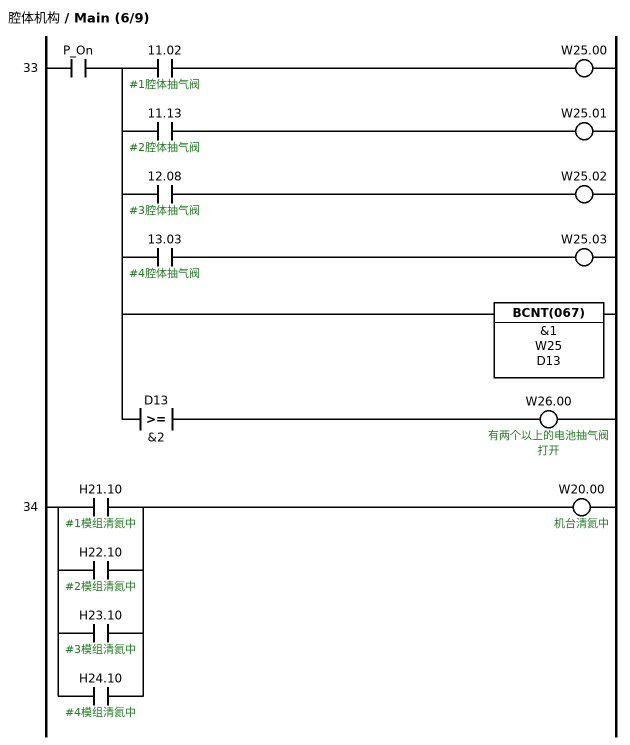
; [picture p240: 腔体机构 / Main, rungs 33-34]
; rung 33
LD P_On
OUT TR0
AND 11.02  ; #1腔体抽气阀
OUT W25.00
LD TR0
AND 11.13  ; #2腔体抽气阀
OUT W25.01
LD TR0
AND 12.08  ; #3腔体抽气阀
OUT W25.02
LD TR0
AND 13.03  ; #4腔体抽气阀
OUT W25.03
LD TR0
BCNT(067) &1 W25 D13
AND>=(325) D13 &2
OUT W26.00  ; 有两个以上的电池抽气阀打开
; rung 34
LD H21.10  ; #1模组清氦中
OR H22.10  ; #2模组清氦中
OR H23.10  ; #3模组清氦中
OR H24.10  ; #4模组清氦中
OUT W20.00  ; 机台清氦中

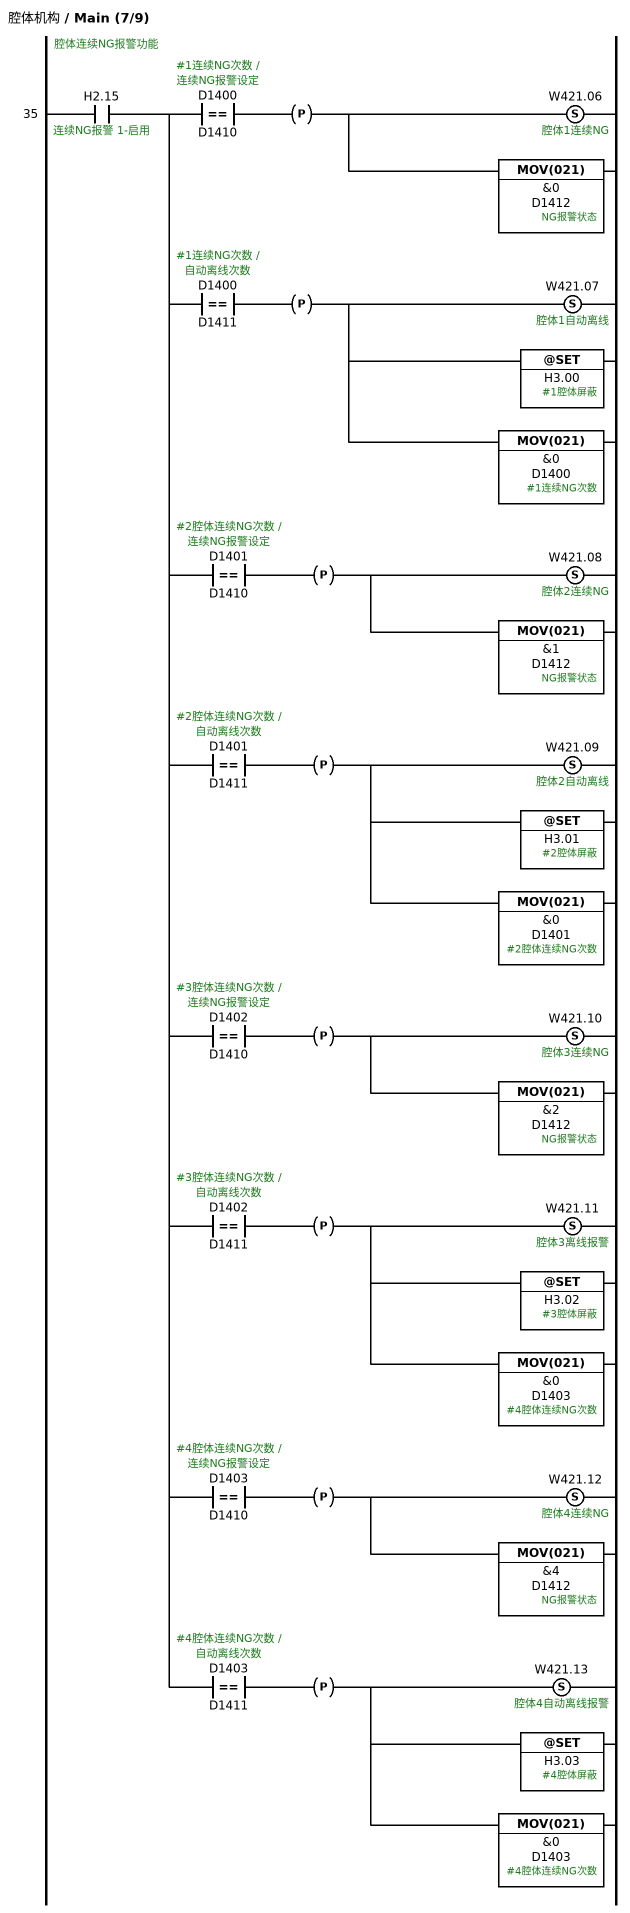
; rung 35: 腔体连续NG报警功能
LD H2.15  ; 连续NG报警 1-启用
OUT TR0
AND=(300) D1400 D1410  ; #1连续NG次数, 连续NG报警设定
UP(521)
SET W421.06  ; 腔体1连续NG
MOV(021) &0 D1412  ; NG报警状态
LD TR0
AND=(300) D1400 D1411  ; #1连续NG次数, 自动离线次数
UP(521)
SET W421.07  ; 腔体1自动离线
@SET H3.00  ; #1腔体屏蔽
MOV(021) &0 D1400  ; #1连续NG次数
LD TR0
AND=(300) D1401 D1410  ; #2腔体连续NG次数, 连续NG报警设定
UP(521)
SET W421.08  ; 腔体2连续NG
MOV(021) &1 D1412  ; NG报警状态
LD TR0
AND=(300) D1401 D1411  ; #2腔体连续NG次数, 自动离线次数
UP(521)
SET W421.09  ; 腔体2自动离线
@SET H3.01  ; #2腔体屏蔽
MOV(021) &0 D1401  ; #2腔体连续NG次数
LD TR0
AND=(300) D1402 D1410  ; #3腔体连续NG次数, 连续NG报警设定
UP(521)
SET W421.10  ; 腔体3连续NG
MOV(021) &2 D1412  ; NG报警状态
LD TR0
AND=(300) D1402 D1411  ; #3腔体连续NG次数, 自动离线次数
UP(521)
SET W421.11  ; 腔体3离线报警
@SET H3.02  ; #3腔体屏蔽
MOV(021) &0 D1403  ; #4腔体连续NG次数
LD TR0
AND=(300) D1403 D1410  ; #4腔体连续NG次数, 连续NG报警设定
UP(521)
SET W421.12  ; 腔体4连续NG
MOV(021) &4 D1412  ; NG报警状态
LD TR0
AND=(300) D1403 D1411  ; #4腔体连续NG次数, 自动离线次数
UP(521)
SET W421.13  ; 腔体4自动离线报警
@SET H3.03  ; #4腔体屏蔽
MOV(021) &0 D1403  ; #4腔体连续NG次数

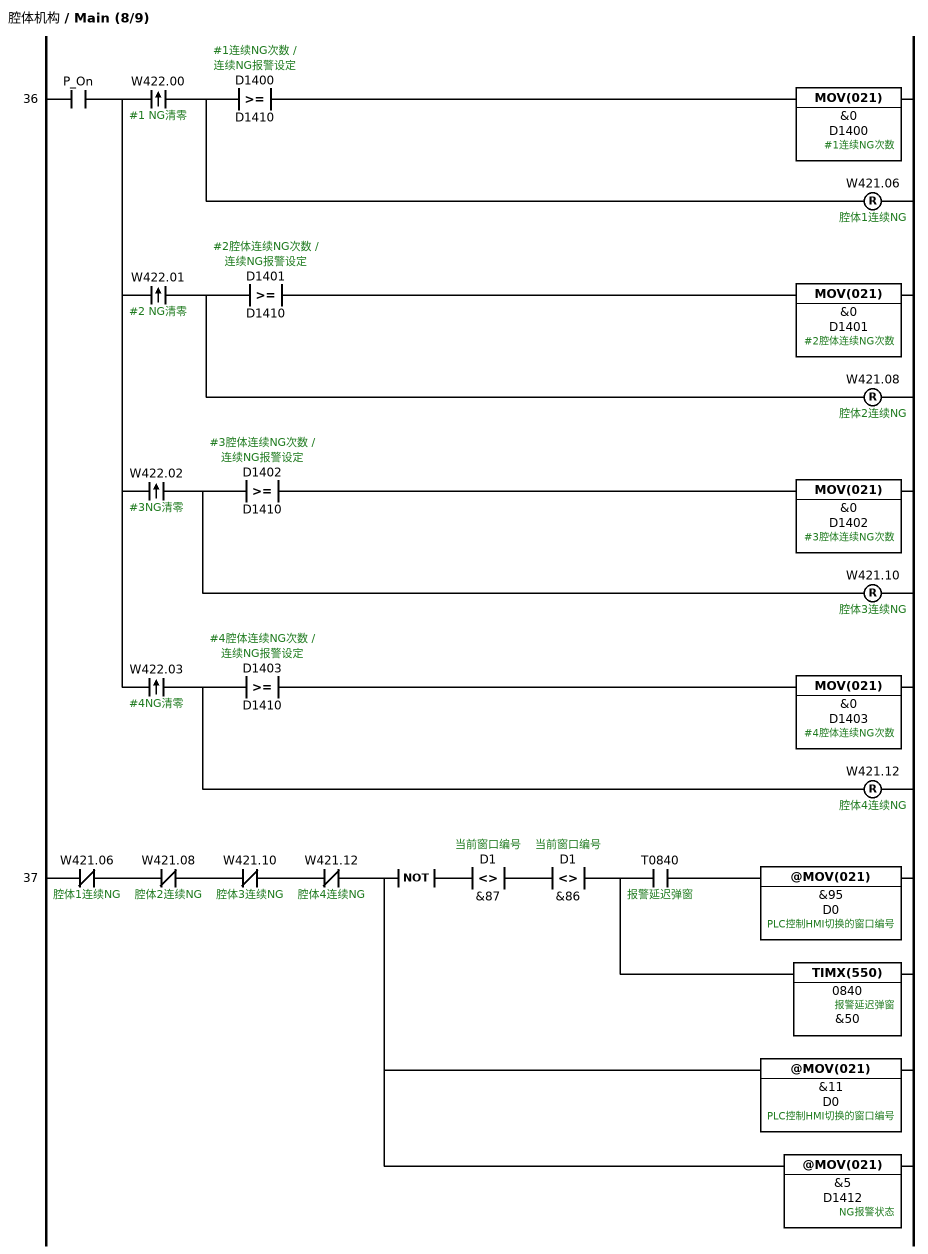
; rung 36
LD P_On
OUT TR0
@AND W422.00  ; #1 NG清零
OUT TR1
AND>=(325) D1400 D1410  ; #1连续NG次数, 连续NG报警设定
MOV(021) &0 D1400  ; #1连续NG次数
LD TR1
RSET W421.06  ; 腔体1连续NG
LD TR0
@AND W422.01  ; #2 NG清零
OUT TR1
AND>=(325) D1401 D1410  ; #2腔体连续NG次数, 连续NG报警设定
MOV(021) &0 D1401  ; #2腔体连续NG次数
LD TR1
RSET W421.08  ; 腔体2连续NG
LD TR0
@AND W422.02  ; #3NG清零
OUT TR1
AND>=(325) D1402 D1410  ; #3腔体连续NG次数, 连续NG报警设定
MOV(021) &0 D1402  ; #3腔体连续NG次数
LD TR1
RSET W421.10  ; 腔体3连续NG
LD TR0
@AND W422.03  ; #4NG清零
OUT TR0
AND>=(325) D1403 D1410  ; #4腔体连续NG次数, 连续NG报警设定
MOV(021) &0 D1403  ; #4腔体连续NG次数
LD TR0
RSET W421.12  ; 腔体4连续NG
; rung 37
LDNOT W421.06  ; 腔体1连续NG
ANDNOT W421.08  ; 腔体2连续NG
ANDNOT W421.10  ; 腔体3连续NG
ANDNOT W421.12  ; 腔体4连续NG
OUT TR0
NOT(520)
AND<>(305) D1 &87  ; 当前窗口编号
AND<>(305) D1 &86  ; 当前窗口编号
OUT TR1
AND T0840  ; 报警延迟弹窗
@MOV(021) &95 D0  ; PLC控制HMI切换的窗口编号
LD TR1
TIMX(550) 0840 &50  ; 报警延迟弹窗
LD TR0
@MOV(021) &11 D0  ; PLC控制HMI切换的窗口编号
@MOV(021) &5 D1412  ; NG报警状态

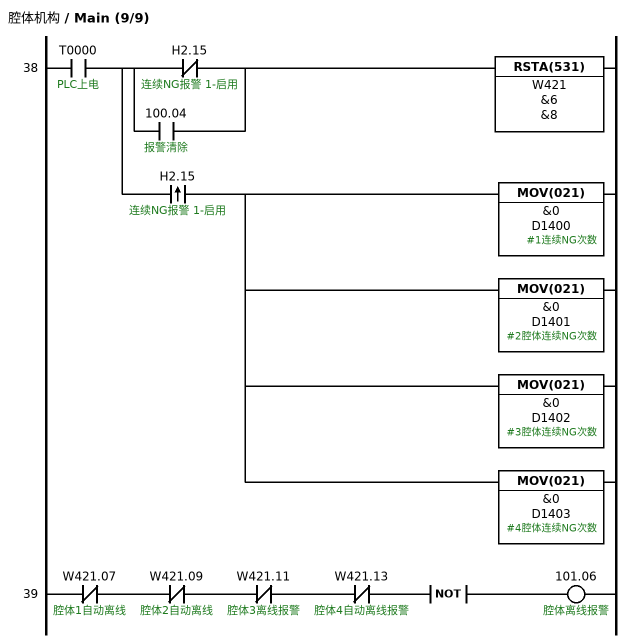
; rung 38
LD T0000  ; PLC上电
OUT TR0
LDNOT H2.15  ; 连续NG报警 1-启用
OR 100.04  ; 报警清除
ANDLD
RSTA(531) W421 &6 &8
LD TR0
@AND H2.15  ; 连续NG报警 1-启用
MOV(021) &0 D1400  ; #1连续NG次数
MOV(021) &0 D1401  ; #2腔体连续NG次数
MOV(021) &0 D1402  ; #3腔体连续NG次数
MOV(021) &0 D1403  ; #4腔体连续NG次数
; rung 39
LDNOT W421.07  ; 腔体1自动离线
ANDNOT W421.09  ; 腔体2自动离线
ANDNOT W421.11  ; 腔体3离线报警
ANDNOT W421.13  ; 腔体4自动离线报警
NOT(520)
OUT 101.06  ; 腔体离线报警

### Section 工站复位

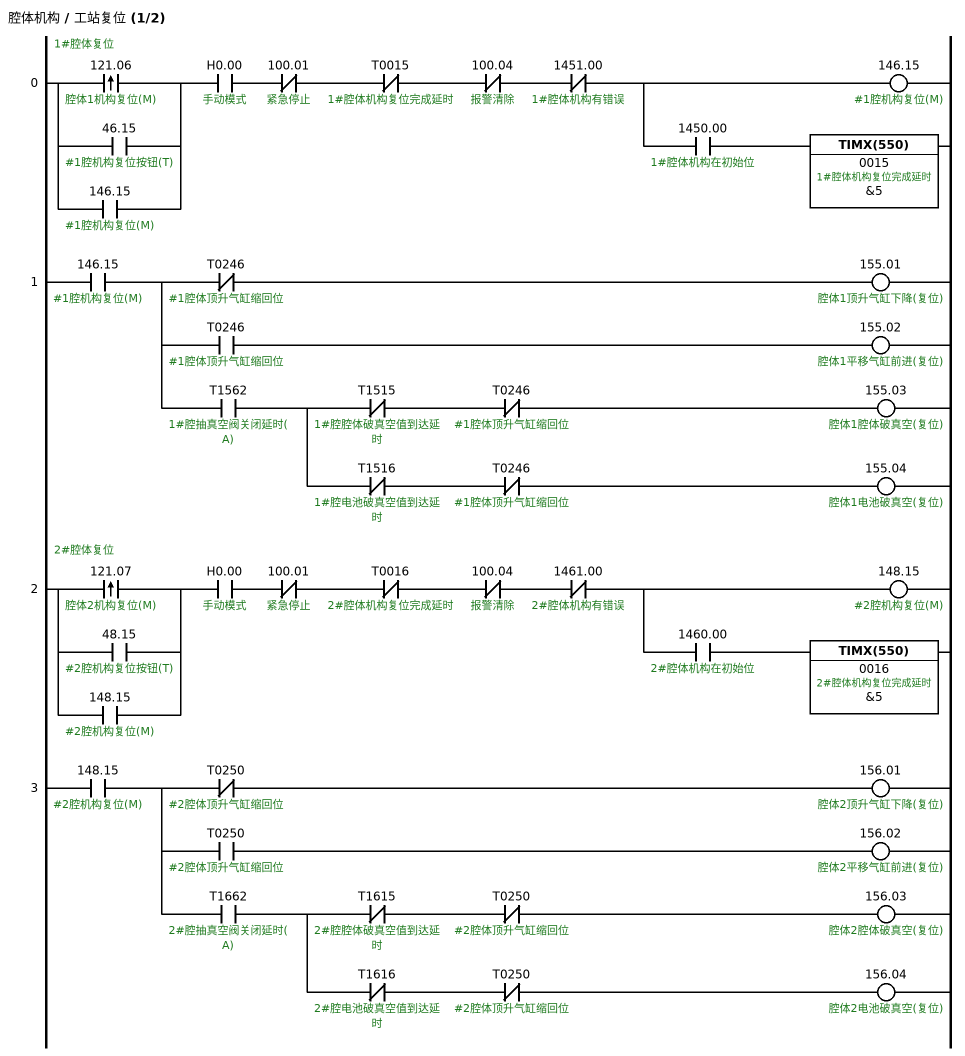
; rung 0: 1#腔体复位
@LD 121.06  ; 腔体1机构复位(M)
OR 46.15  ; #1腔机构复位按钮(T)
OR 146.15  ; #1腔机构复位(M)
AND H0.00  ; 手动模式
ANDNOT 100.01  ; 紧急停止
ANDNOT T0015  ; 1#腔体机构复位完成延时
ANDNOT 100.04  ; 报警清除
ANDNOT 1451.00  ; 1#腔体机构有错误
OUT 146.15  ; #1腔机构复位(M)
AND 1450.00  ; 1#腔体机构在初始位
TIMX(550) 0015 &5  ; 1#腔体机构复位完成延时
; rung 1
LD 146.15  ; #1腔机构复位(M)
OUT TR0
ANDNOT T0246  ; #1腔体顶升气缸缩回位
OUT 155.01  ; 腔体1顶升气缸下降(复位)
LD TR0
AND T0246  ; #1腔体顶升气缸缩回位
OUT 155.02  ; 腔体1平移气缸前进(复位)
LD TR0
AND T1562  ; 1#腔抽真空阀关闭延时(A)
OUT TR0
ANDNOT T1515  ; 1#腔腔体破真空值到达延时
ANDNOT T0246  ; #1腔体顶升气缸缩回位
OUT 155.03  ; 腔体1腔体破真空(复位)
LD TR0
ANDNOT T1516  ; 1#腔电池破真空值到达延时
ANDNOT T0246  ; #1腔体顶升气缸缩回位
OUT 155.04  ; 腔体1电池破真空(复位)
; rung 2: 2#腔体复位
@LD 121.07  ; 腔体2机构复位(M)
OR 48.15  ; #2腔机构复位按钮(T)
OR 148.15  ; #2腔机构复位(M)
AND H0.00  ; 手动模式
ANDNOT 100.01  ; 紧急停止
ANDNOT T0016  ; 2#腔体机构复位完成延时
ANDNOT 100.04  ; 报警清除
ANDNOT 1461.00  ; 2#腔体机构有错误
OUT 148.15  ; #2腔机构复位(M)
AND 1460.00  ; 2#腔体机构在初始位
TIMX(550) 0016 &5  ; 2#腔体机构复位完成延时
; rung 3
LD 148.15  ; #2腔机构复位(M)
OUT TR0
ANDNOT T0250  ; #2腔体顶升气缸缩回位
OUT 156.01  ; 腔体2顶升气缸下降(复位)
LD TR0
AND T0250  ; #2腔体顶升气缸缩回位
OUT 156.02  ; 腔体2平移气缸前进(复位)
LD TR0
AND T1662  ; 2#腔抽真空阀关闭延时(A)
OUT TR0
ANDNOT T1615  ; 2#腔腔体破真空值到达延时
ANDNOT T0250  ; #2腔体顶升气缸缩回位
OUT 156.03  ; 腔体2腔体破真空(复位)
LD TR0
ANDNOT T1616  ; 2#腔电池破真空值到达延时
ANDNOT T0250  ; #2腔体顶升气缸缩回位
OUT 156.04  ; 腔体2电池破真空(复位)

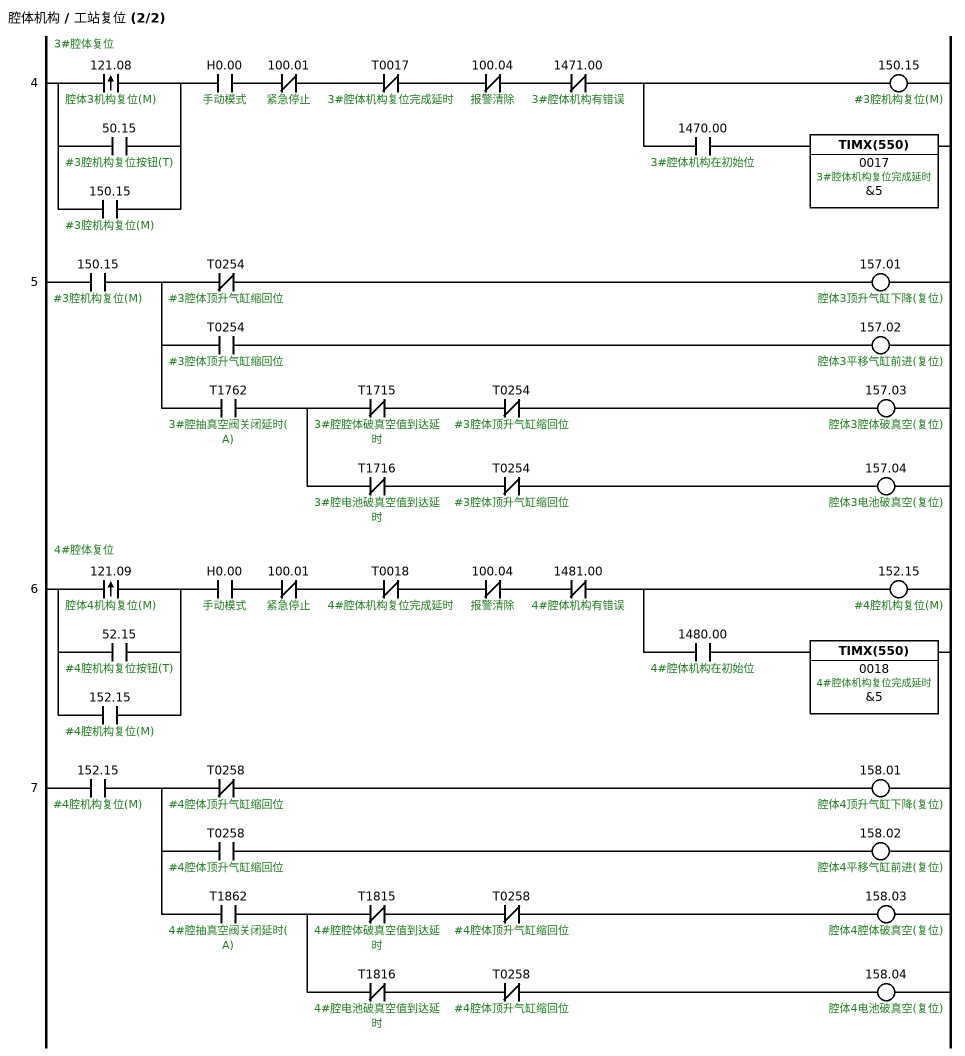
; rung 4: 3#腔体复位
@LD 121.08  ; 腔体3机构复位(M)
OR 50.15  ; #3腔机构复位按钮(T)
OR 150.15  ; #3腔机构复位(M)
AND H0.00  ; 手动模式
ANDNOT 100.01  ; 紧急停止
ANDNOT T0017  ; 3#腔体机构复位完成延时
ANDNOT 100.04  ; 报警清除
ANDNOT 1471.00  ; 3#腔体机构有错误
OUT 150.15  ; #3腔机构复位(M)
AND 1470.00  ; 3#腔体机构在初始位
TIMX(550) 0017 &5  ; 3#腔体机构复位完成延时
; rung 5
LD 150.15  ; #3腔机构复位(M)
OUT TR0
ANDNOT T0254  ; #3腔体顶升气缸缩回位
OUT 157.01  ; 腔体3顶升气缸下降(复位)
LD TR0
AND T0254  ; #3腔体顶升气缸缩回位
OUT 157.02  ; 腔体3平移气缸前进(复位)
LD TR0
AND T1762  ; 3#腔抽真空阀关闭延时(A)
OUT TR0
ANDNOT T1715  ; 3#腔腔体破真空值到达延时
ANDNOT T0254  ; #3腔体顶升气缸缩回位
OUT 157.03  ; 腔体3腔体破真空(复位)
LD TR0
ANDNOT T1716  ; 3#腔电池破真空值到达延时
ANDNOT T0254  ; #3腔体顶升气缸缩回位
OUT 157.04  ; 腔体3电池破真空(复位)
; rung 6: 4#腔体复位
@LD 121.09  ; 腔体4机构复位(M)
OR 52.15  ; #4腔机构复位按钮(T)
OR 152.15  ; #4腔机构复位(M)
AND H0.00  ; 手动模式
ANDNOT 100.01  ; 紧急停止
ANDNOT T0018  ; 4#腔体机构复位完成延时
ANDNOT 100.04  ; 报警清除
ANDNOT 1481.00  ; 4#腔体机构有错误
OUT 152.15  ; #4腔机构复位(M)
AND 1480.00  ; 4#腔体机构在初始位
TIMX(550) 0018 &5  ; 4#腔体机构复位完成延时
; rung 7
LD 152.15  ; #4腔机构复位(M)
OUT TR0
ANDNOT T0258  ; #4腔体顶升气缸缩回位
OUT 158.01  ; 腔体4顶升气缸下降(复位)
LD TR0
AND T0258  ; #4腔体顶升气缸缩回位
OUT 158.02  ; 腔体4平移气缸前进(复位)
LD TR0
AND T1862  ; 4#腔抽真空阀关闭延时(A)
OUT TR0
ANDNOT T1815  ; 4#腔腔体破真空值到达延时
ANDNOT T0258  ; #4腔体顶升气缸缩回位
OUT 158.03  ; 腔体4腔体破真空(复位)
LD TR0
ANDNOT T1816  ; 4#腔电池破真空值到达延时
ANDNOT T0258  ; #4腔体顶升气缸缩回位
OUT 158.04  ; 腔体4电池破真空(复位)

### Section _1_腔体手动

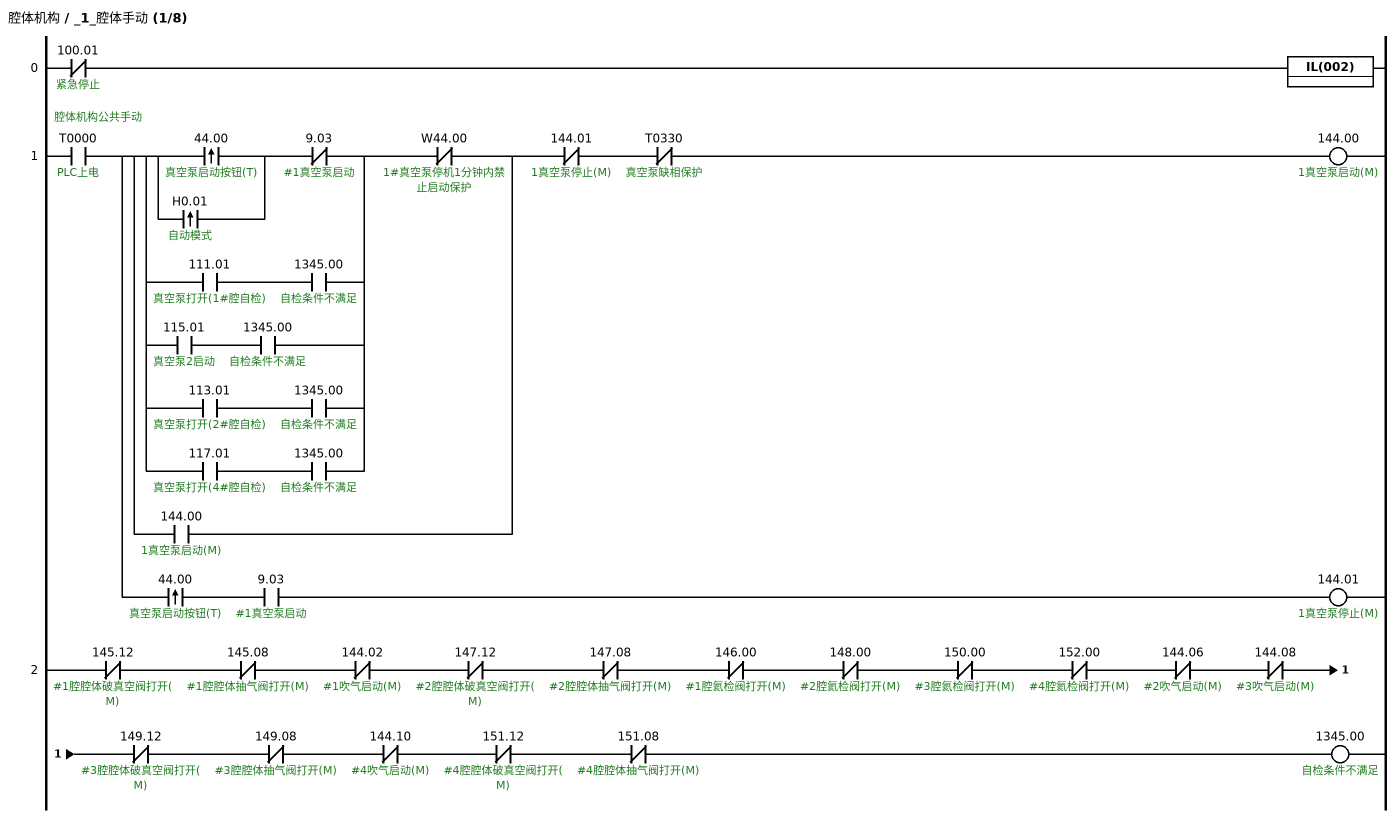
; rung 0
LDNOT 100.01  ; 紧急停止
IL(002)
; rung 1: 腔体机构公共手动
LD T0000  ; PLC上电
OUT TR0
@LD 44.00  ; 真空泵启动按钮(T)
@OR H0.01  ; 自动模式
ANDNOT 9.03  ; #1真空泵启动
LD 111.01  ; 真空泵打开(1#腔自检)
AND 1345.00  ; 自检条件不满足
ORLD
LD 115.01  ; 真空泵2启动
AND 1345.00  ; 自检条件不满足
ORLD
LD 113.01  ; 真空泵打开(2#腔自检)
AND 1345.00  ; 自检条件不满足
ORLD
LD 117.01  ; 真空泵打开(4#腔自检)
AND 1345.00  ; 自检条件不满足
ORLD
ANDNOT W44.00  ; 1#真空泵停机1分钟内禁止启动保护
OR 144.00  ; 1真空泵启动(M)
ANDLD
ANDNOT 144.01  ; 1真空泵停止(M)
ANDNOT T0330  ; 真空泵缺相保护
OUT 144.00  ; 1真空泵启动(M)
LD TR0
@AND 44.00  ; 真空泵启动按钮(T)
AND 9.03  ; #1真空泵启动
OUT 144.01  ; 1真空泵停止(M)
; rung 2
LDNOT 145.12  ; #1腔腔体破真空阀打开(M)
ANDNOT 145.08  ; #1腔腔体抽气阀打开(M)
ANDNOT 144.02  ; #1吹气启动(M)
ANDNOT 147.12  ; #2腔腔体破真空阀打开(M)
ANDNOT 147.08  ; #2腔腔体抽气阀打开(M)
ANDNOT 146.00  ; #1腔氦检阀打开(M)
ANDNOT 148.00  ; #2腔氦检阀打开(M)
ANDNOT 150.00  ; #3腔氦检阀打开(M)
ANDNOT 152.00  ; #4腔氦检阀打开(M)
ANDNOT 144.06  ; #2吹气启动(M)
ANDNOT 144.08  ; #3吹气启动(M)
ANDNOT 149.12  ; #3腔腔体破真空阀打开(M)
ANDNOT 149.08  ; #3腔腔体抽气阀打开(M)
ANDNOT 144.10  ; #4吹气启动(M)
ANDNOT 151.12  ; #4腔腔体破真空阀打开(M)
ANDNOT 151.08  ; #4腔腔体抽气阀打开(M)
OUT 1345.00  ; 自检条件不满足

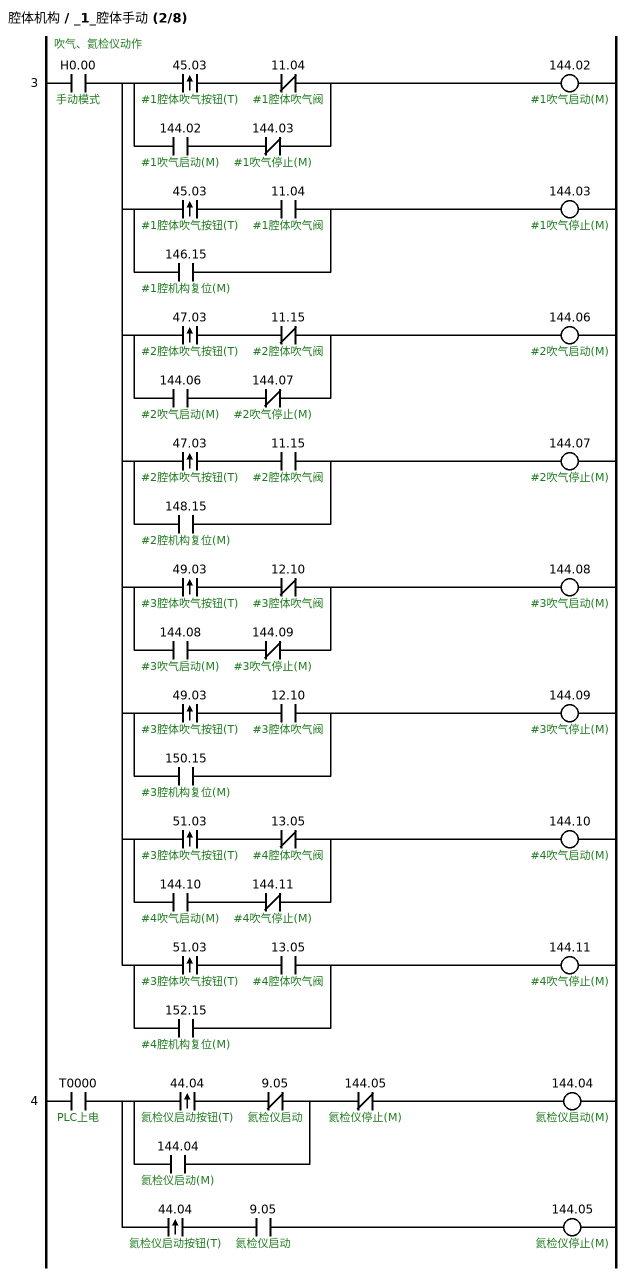
; rung 3: 吹气、氦检仪动作
LD H0.00  ; 手动模式
OUT TR0
@LD 45.03  ; #1腔体吹气按钮(T)
ANDNOT 11.04  ; #1腔体吹气阀
LD 144.02  ; #1吹气启动(M)
ANDNOT 144.03  ; #1吹气停止(M)
ORLD
ANDLD
OUT 144.02  ; #1吹气启动(M)
LD TR0
@LD 45.03  ; #1腔体吹气按钮(T)
AND 11.04  ; #1腔体吹气阀
OR 146.15  ; #1腔机构复位(M)
ANDLD
OUT 144.03  ; #1吹气停止(M)
LD TR0
@LD 47.03  ; #2腔体吹气按钮(T)
ANDNOT 11.15  ; #2腔体吹气阀
LD 144.06  ; #2吹气启动(M)
ANDNOT 144.07  ; #2吹气停止(M)
ORLD
ANDLD
OUT 144.06  ; #2吹气启动(M)
LD TR0
@LD 47.03  ; #2腔体吹气按钮(T)
AND 11.15  ; #2腔体吹气阀
OR 148.15  ; #2腔机构复位(M)
ANDLD
OUT 144.07  ; #2吹气停止(M)
LD TR0
@LD 49.03  ; #3腔体吹气按钮(T)
ANDNOT 12.10  ; #3腔体吹气阀
LD 144.08  ; #3吹气启动(M)
ANDNOT 144.09  ; #3吹气停止(M)
ORLD
ANDLD
OUT 144.08  ; #3吹气启动(M)
LD TR0
@LD 49.03  ; #3腔体吹气按钮(T)
AND 12.10  ; #3腔体吹气阀
OR 150.15  ; #3腔机构复位(M)
ANDLD
OUT 144.09  ; #3吹气停止(M)
LD TR0
@LD 51.03  ; #3腔体吹气按钮(T)
ANDNOT 13.05  ; #4腔体吹气阀
LD 144.10  ; #4吹气启动(M)
ANDNOT 144.11  ; #4吹气停止(M)
ORLD
ANDLD
OUT 144.10  ; #4吹气启动(M)
LD TR0
@LD 51.03  ; #3腔体吹气按钮(T)
AND 13.05  ; #4腔体吹气阀
OR 152.15  ; #4腔机构复位(M)
ANDLD
OUT 144.11  ; #4吹气停止(M)
; rung 4
LD T0000  ; PLC上电
OUT TR0
@LD 44.04  ; 氦检仪启动按钮(T)
ANDNOT 9.05  ; 氦检仪启动
OR 144.04  ; 氦检仪启动(M)
ANDLD
ANDNOT 144.05  ; 氦检仪停止(M)
OUT 144.04  ; 氦检仪启动(M)
LD TR0
@AND 44.04  ; 氦检仪启动按钮(T)
AND 9.05  ; 氦检仪启动
OUT 144.05  ; 氦检仪停止(M)

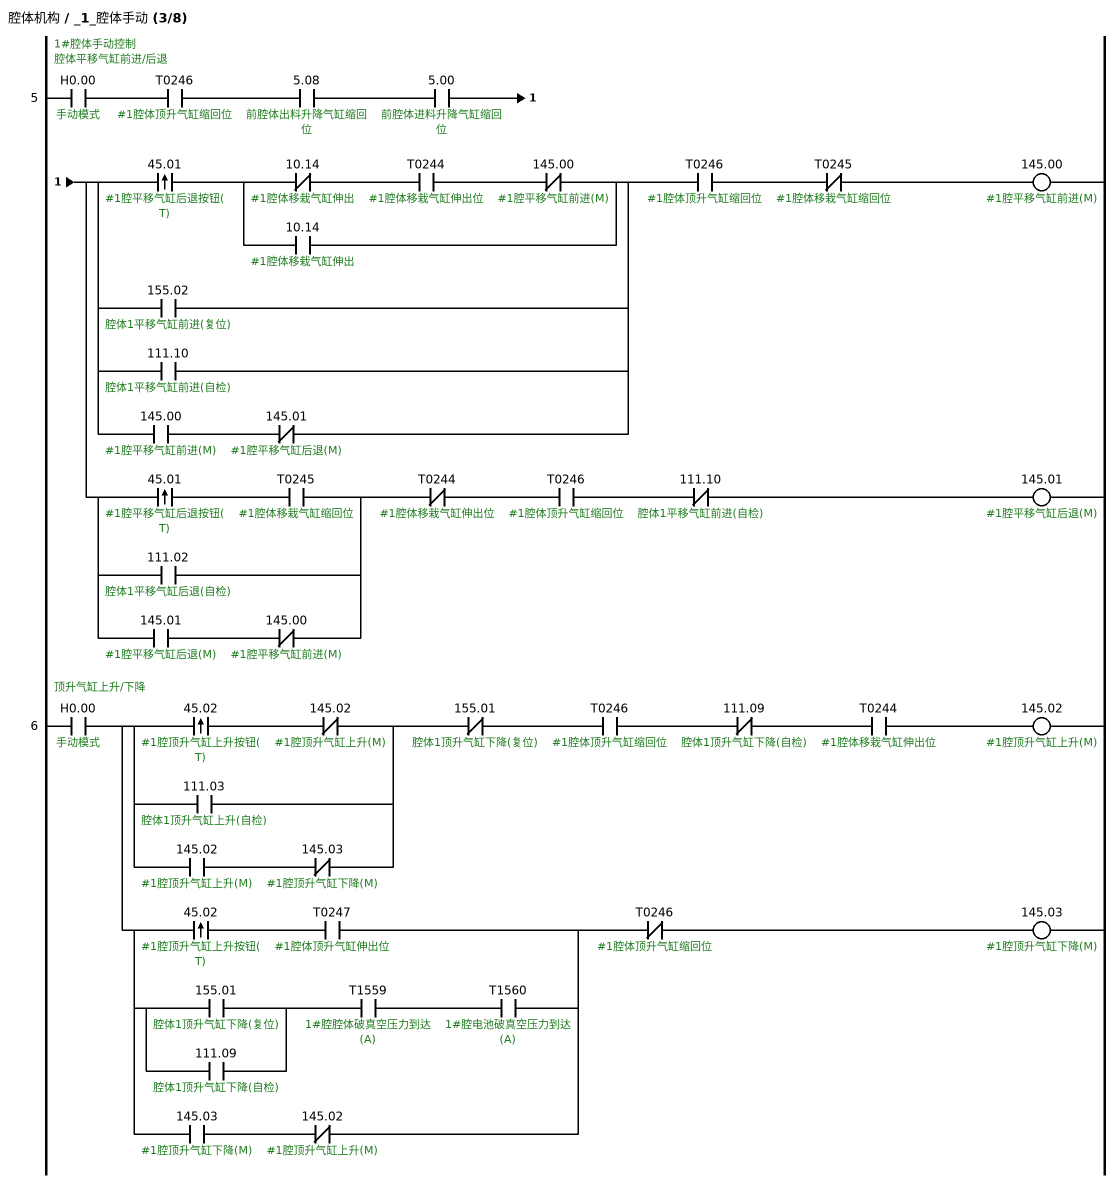
; rung 5: 1#腔体手动控制 / 腔体平移气缸前进/后退
LD H0.00  ; 手动模式
AND T0246  ; #1腔体顶升气缸缩回位
AND 5.08  ; 前腔体出料升降气缸缩回位
AND 5.00  ; 前腔体进料升降气缸缩回位
OUT TR0
@LD 45.01  ; #1腔平移气缸后退按钮(T)
LDNOT 10.14  ; #1腔体移栽气缸伸出
AND T0244  ; #1腔体移栽气缸伸出位
ANDNOT 145.00  ; #1腔平移气缸前进(M)
OR 10.14  ; #1腔体移栽气缸伸出
ANDLD
OR 155.02  ; 腔体1平移气缸前进(复位)
OR 111.10  ; 腔体1平移气缸前进(自检)
LD 145.00  ; #1腔平移气缸前进(M)
ANDNOT 145.01  ; #1腔平移气缸后退(M)
ORLD
ANDLD
AND T0246  ; #1腔体顶升气缸缩回位
ANDNOT T0245  ; #1腔体移栽气缸缩回位
OUT 145.00  ; #1腔平移气缸前进(M)
LD TR0
@LD 45.01  ; #1腔平移气缸后退按钮(T)
AND T0245  ; #1腔体移栽气缸缩回位
OR 111.02  ; 腔体1平移气缸后退(自检)
LD 145.01  ; #1腔平移气缸后退(M)
ANDNOT 145.00  ; #1腔平移气缸前进(M)
ORLD
ANDLD
ANDNOT T0244  ; #1腔体移栽气缸伸出位
AND T0246  ; #1腔体顶升气缸缩回位
ANDNOT 111.10  ; 腔体1平移气缸前进(自检)
OUT 145.01  ; #1腔平移气缸后退(M)
; rung 6: 顶升气缸上升/下降
LD H0.00  ; 手动模式
OUT TR0
@LD 45.02  ; #1腔顶升气缸上升按钮(T)
ANDNOT 145.02  ; #1腔顶升气缸上升(M)
OR 111.03  ; 腔体1顶升气缸上升(自检)
LD 145.02  ; #1腔顶升气缸上升(M)
ANDNOT 145.03  ; #1腔顶升气缸下降(M)
ORLD
ANDLD
ANDNOT 155.01  ; 腔体1顶升气缸下降(复位)
AND T0246  ; #1腔体顶升气缸缩回位
ANDNOT 111.09  ; 腔体1顶升气缸下降(自检)
AND T0244  ; #1腔体移栽气缸伸出位
OUT 145.02  ; #1腔顶升气缸上升(M)
LD TR0
@LD 45.02  ; #1腔顶升气缸上升按钮(T)
AND T0247  ; #1腔体顶升气缸伸出位
LD 155.01  ; 腔体1顶升气缸下降(复位)
OR 111.09  ; 腔体1顶升气缸下降(自检)
AND T1559  ; 1#腔腔体破真空压力到达(A)
AND T1560  ; 1#腔电池破真空压力到达(A)
ORLD
LD 145.03  ; #1腔顶升气缸下降(M)
ANDNOT 145.02  ; #1腔顶升气缸上升(M)
ORLD
ANDLD
ANDNOT T0246  ; #1腔体顶升气缸缩回位
OUT 145.03  ; #1腔顶升气缸下降(M)

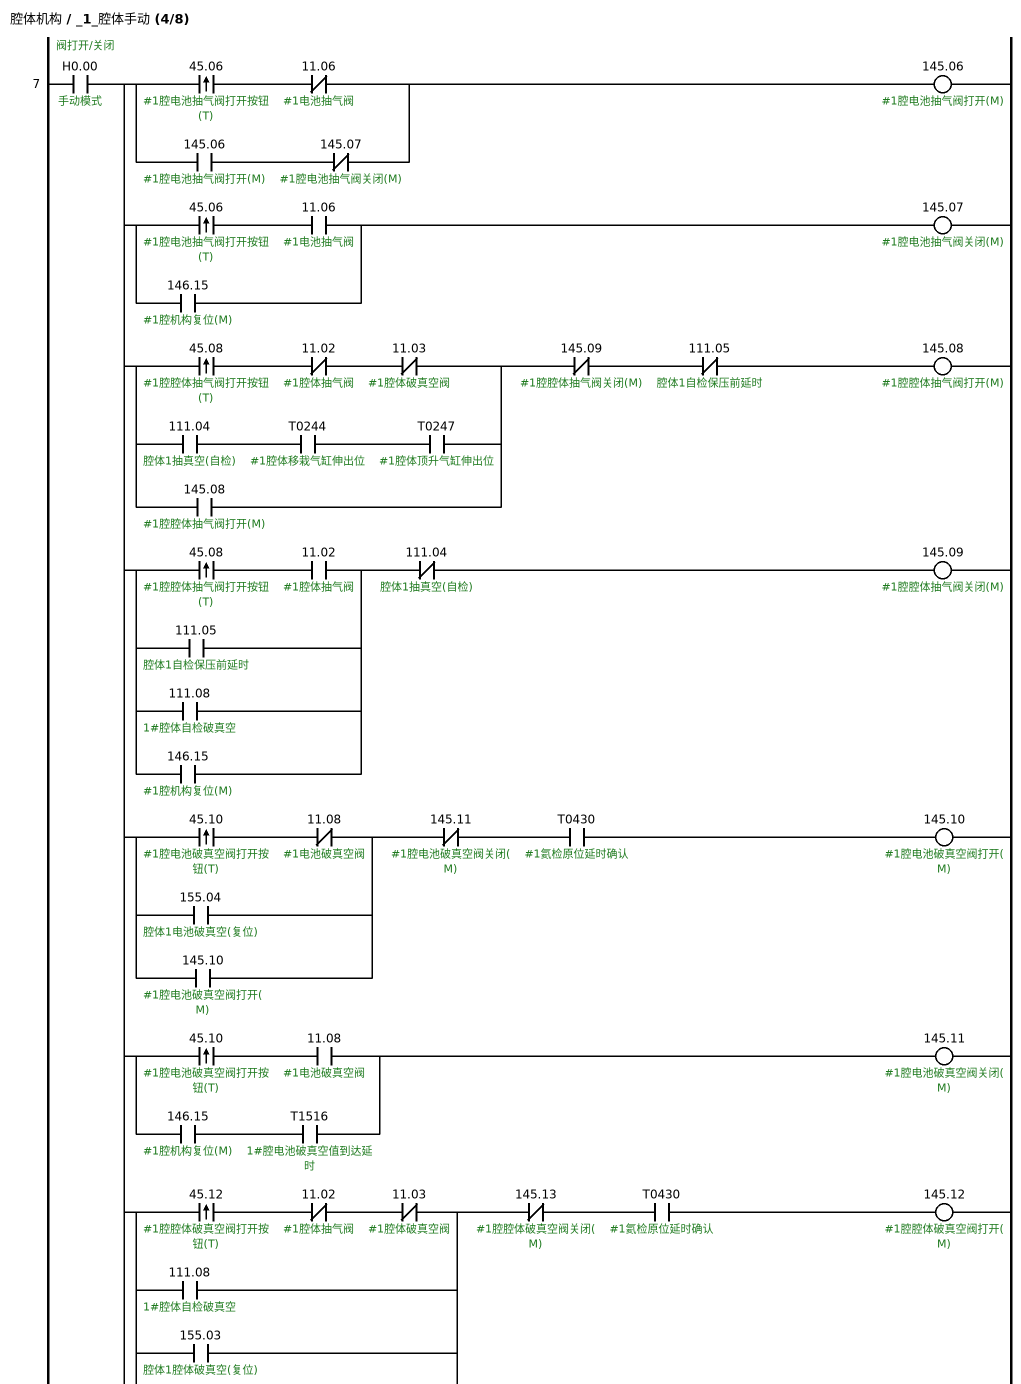

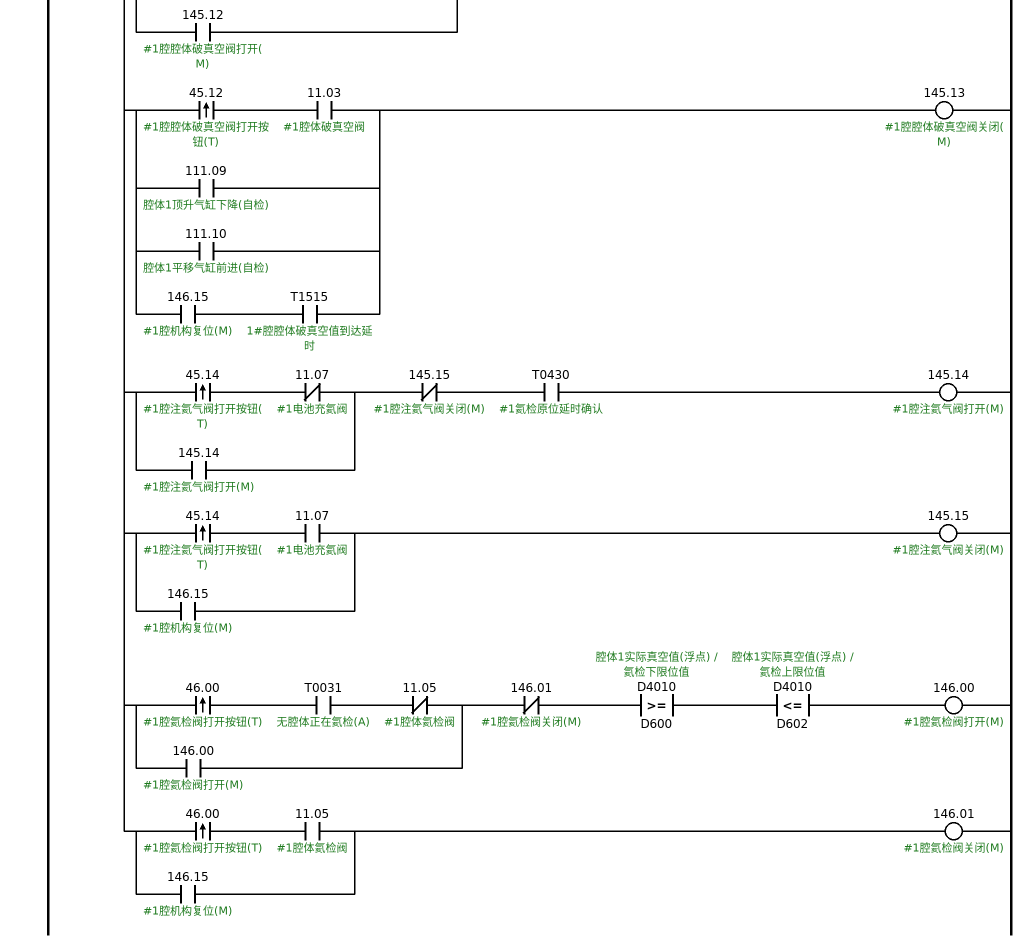
; rung 7: 阀打开/关闭
LD H0.00  ; 手动模式
OUT TR0
@LD 45.06  ; #1腔电池抽气阀打开按钮(T)
ANDNOT 11.06  ; #1电池抽气阀
LD 145.06  ; #1腔电池抽气阀打开(M)
ANDNOT 145.07  ; #1腔电池抽气阀关闭(M)
ORLD
ANDLD
OUT 145.06  ; #1腔电池抽气阀打开(M)
LD TR0
@LD 45.06  ; #1腔电池抽气阀打开按钮(T)
AND 11.06  ; #1电池抽气阀
OR 146.15  ; #1腔机构复位(M)
ANDLD
OUT 145.07  ; #1腔电池抽气阀关闭(M)
LD TR0
@LD 45.08  ; #1腔腔体抽气阀打开按钮(T)
ANDNOT 11.02  ; #1腔体抽气阀
ANDNOT 11.03  ; #1腔体破真空阀
LD 111.04  ; 腔体1抽真空(自检)
AND T0244  ; #1腔体移栽气缸伸出位
AND T0247  ; #1腔体顶升气缸伸出位
ORLD
OR 145.08  ; #1腔腔体抽气阀打开(M)
ANDLD
ANDNOT 145.09  ; #1腔腔体抽气阀关闭(M)
ANDNOT 111.05  ; 腔体1自检保压前延时
OUT 145.08  ; #1腔腔体抽气阀打开(M)
LD TR0
@LD 45.08  ; #1腔腔体抽气阀打开按钮(T)
AND 11.02  ; #1腔体抽气阀
OR 111.05  ; 腔体1自检保压前延时
OR 111.08  ; 1#腔体自检破真空
OR 146.15  ; #1腔机构复位(M)
ANDLD
ANDNOT 111.04  ; 腔体1抽真空(自检)
OUT 145.09  ; #1腔腔体抽气阀关闭(M)
LD TR0
@LD 45.10  ; #1腔电池破真空阀打开按钮(T)
ANDNOT 11.08  ; #1电池破真空阀
OR 155.04  ; 腔体1电池破真空(复位)
OR 145.10  ; #1腔电池破真空阀打开(M)
ANDLD
ANDNOT 145.11  ; #1腔电池破真空阀关闭(M)
AND T0430  ; #1氦检原位延时确认
OUT 145.10  ; #1腔电池破真空阀打开(M)
LD TR0
@LD 45.10  ; #1腔电池破真空阀打开按钮(T)
AND 11.08  ; #1电池破真空阀
LD 146.15  ; #1腔机构复位(M)
AND T1516  ; 1#腔电池破真空值到达延时
ORLD
ANDLD
OUT 145.11  ; #1腔电池破真空阀关闭(M)
LD TR0
@LD 45.12  ; #1腔腔体破真空阀打开按钮(T)
ANDNOT 11.02  ; #1腔体抽气阀
ANDNOT 11.03  ; #1腔体破真空阀
OR 111.08  ; 1#腔体自检破真空
OR 155.03  ; 腔体1腔体破真空(复位)
OR 145.12  ; #1腔腔体破真空阀打开(M)
ANDLD
ANDNOT 145.13  ; #1腔腔体破真空阀关闭(M)
AND T0430  ; #1氦检原位延时确认
OUT 145.12  ; #1腔腔体破真空阀打开(M)
LD TR0
@LD 45.12  ; #1腔腔体破真空阀打开按钮(T)
AND 11.03  ; #1腔体破真空阀
OR 111.09  ; 腔体1顶升气缸下降(自检)
OR 111.10  ; 腔体1平移气缸前进(自检)
LD 146.15  ; #1腔机构复位(M)
AND T1515  ; 1#腔腔体破真空值到达延时
ORLD
ANDLD
OUT 145.13  ; #1腔腔体破真空阀关闭(M)
LD TR0
@LD 45.14  ; #1腔注氦气阀打开按钮(T)
ANDNOT 11.07  ; #1电池充氦阀
OR 145.14  ; #1腔注氦气阀打开(M)
ANDLD
ANDNOT 145.15  ; #1腔注氦气阀关闭(M)
AND T0430  ; #1氦检原位延时确认
OUT 145.14  ; #1腔注氦气阀打开(M)
LD TR0
@LD 45.14  ; #1腔注氦气阀打开按钮(T)
AND 11.07  ; #1电池充氦阀
OR 146.15  ; #1腔机构复位(M)
ANDLD
OUT 145.15  ; #1腔注氦气阀关闭(M)
LD TR0
@LD 46.00  ; #1腔氦检阀打开按钮(T)
AND T0031  ; 无腔体正在氦检(A)
ANDNOT 11.05  ; #1腔体氦检阀
OR 146.00  ; #1腔氦检阀打开(M)
ANDLD
ANDNOT 146.01  ; #1腔氦检阀关闭(M)
AND>=F(334) D4010 D600  ; 腔体1实际真空值(浮点), 氦检下限位值
AND<=F(332) D4010 D602  ; 腔体1实际真空值(浮点), 氦检上限位值
OUT 146.00  ; #1腔氦检阀打开(M)
LD TR0
@LD 46.00  ; #1腔氦检阀打开按钮(T)
AND 11.05  ; #1腔体氦检阀
OR 146.15  ; #1腔机构复位(M)
ANDLD
OUT 146.01  ; #1腔氦检阀关闭(M)

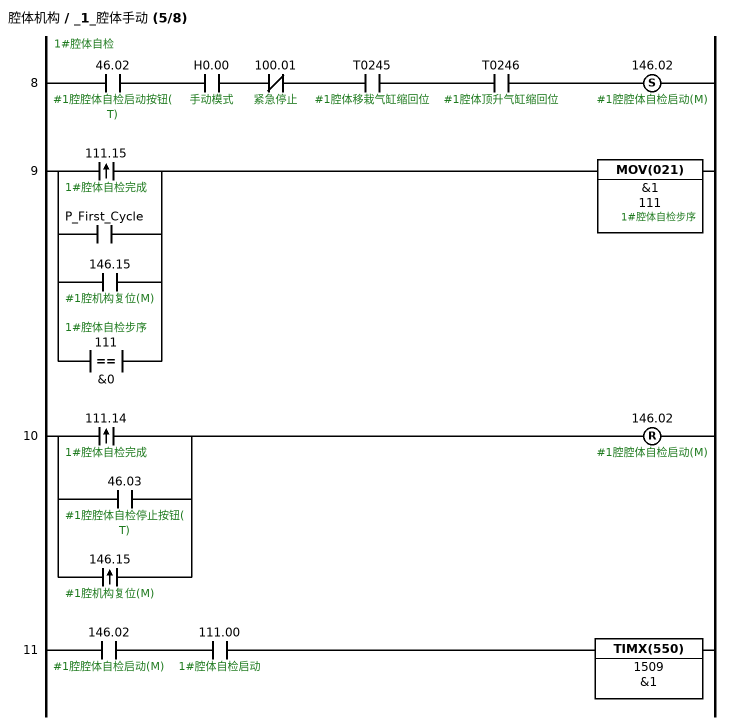
; rung 8: 1#腔体自检
LD 46.02  ; #1腔腔体自检启动按钮(T)
AND H0.00  ; 手动模式
ANDNOT 100.01  ; 紧急停止
AND T0245  ; #1腔体移栽气缸缩回位
AND T0246  ; #1腔体顶升气缸缩回位
SET 146.02  ; #1腔腔体自检启动(M)
; rung 9
@LD 111.15  ; 1#腔体自检完成
OR P_First_Cycle
OR 146.15  ; #1腔机构复位(M)
OR=(300) 111 &0  ; 1#腔体自检步序
MOV(021) &1 111  ; 1#腔体自检步序
; rung 10
@LD 111.14  ; 1#腔体自检完成
OR 46.03  ; #1腔腔体自检停止按钮(T)
@OR 146.15  ; #1腔机构复位(M)
RSET 146.02  ; #1腔腔体自检启动(M)
; rung 11
LD 146.02  ; #1腔腔体自检启动(M)
AND 111.00  ; 1#腔体自检启动
TIMX(550) 1509 &1

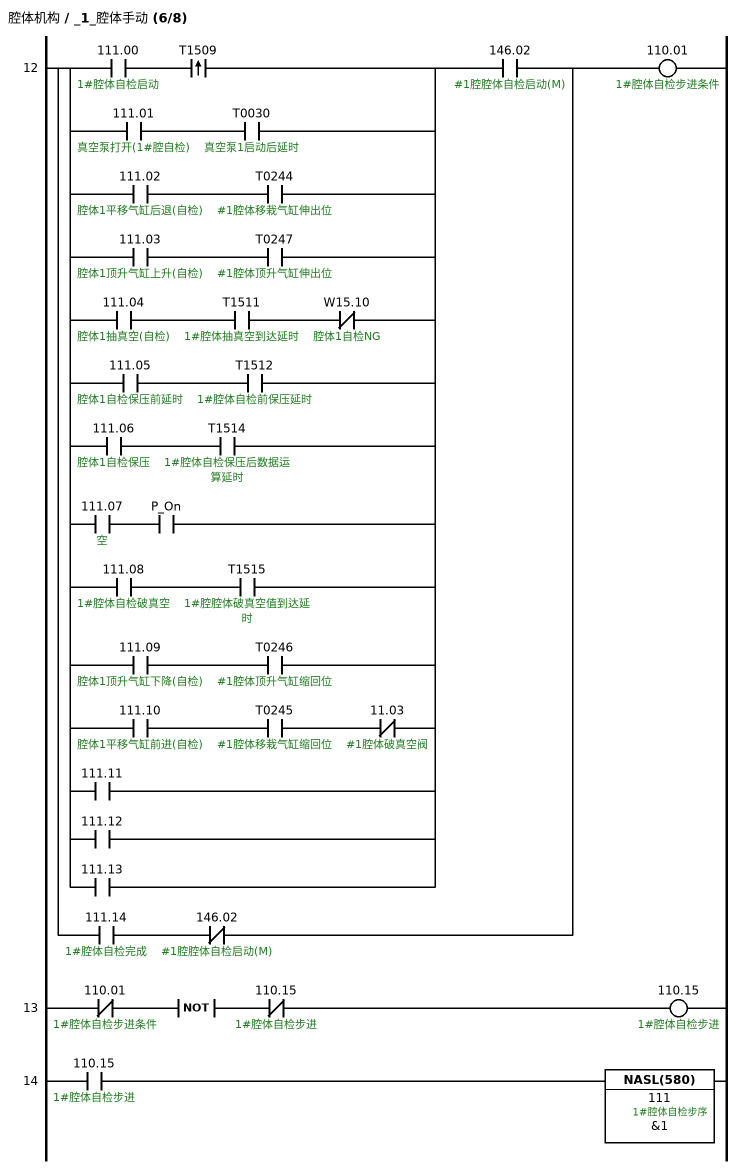
; rung 12
LD 111.00  ; 1#腔体自检启动
@AND T1509
LD 111.01  ; 真空泵打开(1#腔自检)
AND T0030  ; 真空泵1启动后延时
ORLD
LD 111.02  ; 腔体1平移气缸后退(自检)
AND T0244  ; #1腔体移栽气缸伸出位
ORLD
LD 111.03  ; 腔体1顶升气缸上升(自检)
AND T0247  ; #1腔体顶升气缸伸出位
ORLD
LD 111.04  ; 腔体1抽真空(自检)
AND T1511  ; 1#腔体抽真空到达延时
ANDNOT W15.10  ; 腔体1自检NG
ORLD
LD 111.05  ; 腔体1自检保压前延时
AND T1512  ; 1#腔体自检前保压延时
ORLD
LD 111.06  ; 腔体1自检保压
AND T1514  ; 1#腔体自检保压后数据运算延时
ORLD
LD 111.07  ; 空
AND P_On
ORLD
LD 111.08  ; 1#腔体自检破真空
AND T1515  ; 1#腔腔体破真空值到达延时
ORLD
LD 111.09  ; 腔体1顶升气缸下降(自检)
AND T0246  ; #1腔体顶升气缸缩回位
ORLD
LD 111.10  ; 腔体1平移气缸前进(自检)
AND T0245  ; #1腔体移栽气缸缩回位
ANDNOT 11.03  ; #1腔体破真空阀
ORLD
OR 111.11
OR 111.12
OR 111.13
AND 146.02  ; #1腔腔体自检启动(M)
LD 111.14  ; 1#腔体自检完成
ANDNOT 146.02  ; #1腔腔体自检启动(M)
ORLD
OUT 110.01  ; 1#腔体自检步进条件
; rung 13
LDNOT 110.01  ; 1#腔体自检步进条件
NOT(520)
ANDNOT 110.15  ; 1#腔体自检步进
OUT 110.15  ; 1#腔体自检步进
; rung 14
LD 110.15  ; 1#腔体自检步进
NASL(580) 111 &1  ; 1#腔体自检步序

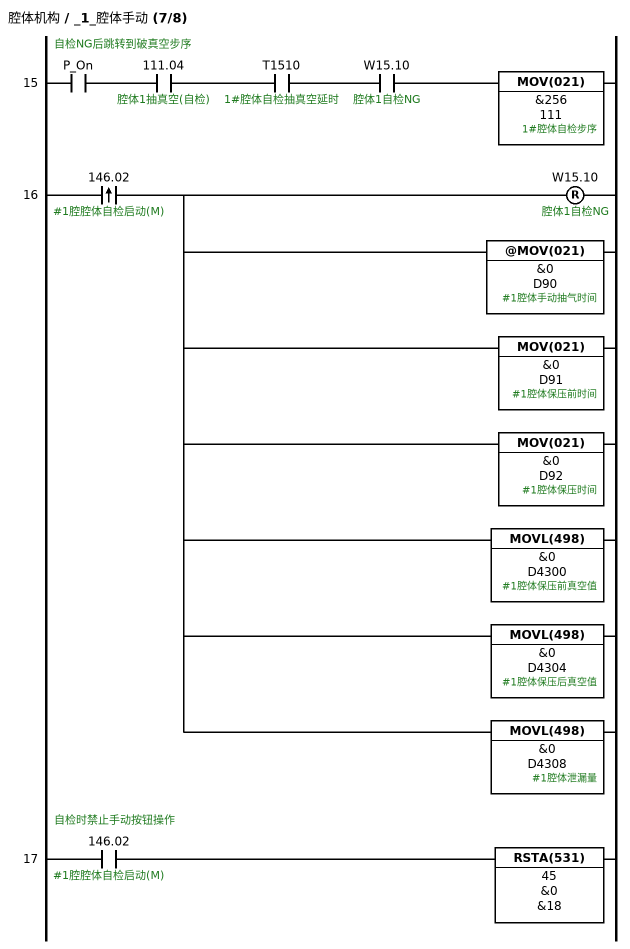
; rung 15: 自检NG后跳转到破真空步序
LD P_On
AND 111.04  ; 腔体1抽真空(自检)
AND T1510  ; 1#腔体自检抽真空延时
AND W15.10  ; 腔体1自检NG
MOV(021) &256 111  ; 1#腔体自检步序
; rung 16
@LD 146.02  ; #1腔腔体自检启动(M)
RSET W15.10  ; 腔体1自检NG
@MOV(021) &0 D90  ; #1腔体手动抽气时间
MOV(021) &0 D91  ; #1腔体保压前时间
MOV(021) &0 D92  ; #1腔体保压时间
MOVL(498) &0 D4300  ; #1腔体保压前真空值
MOVL(498) &0 D4304  ; #1腔体保压后真空值
MOVL(498) &0 D4308  ; #1腔体泄漏量
; rung 17: 自检时禁止手动按钮操作
LD 146.02  ; #1腔腔体自检启动(M)
RSTA(531) 45 &0 &18

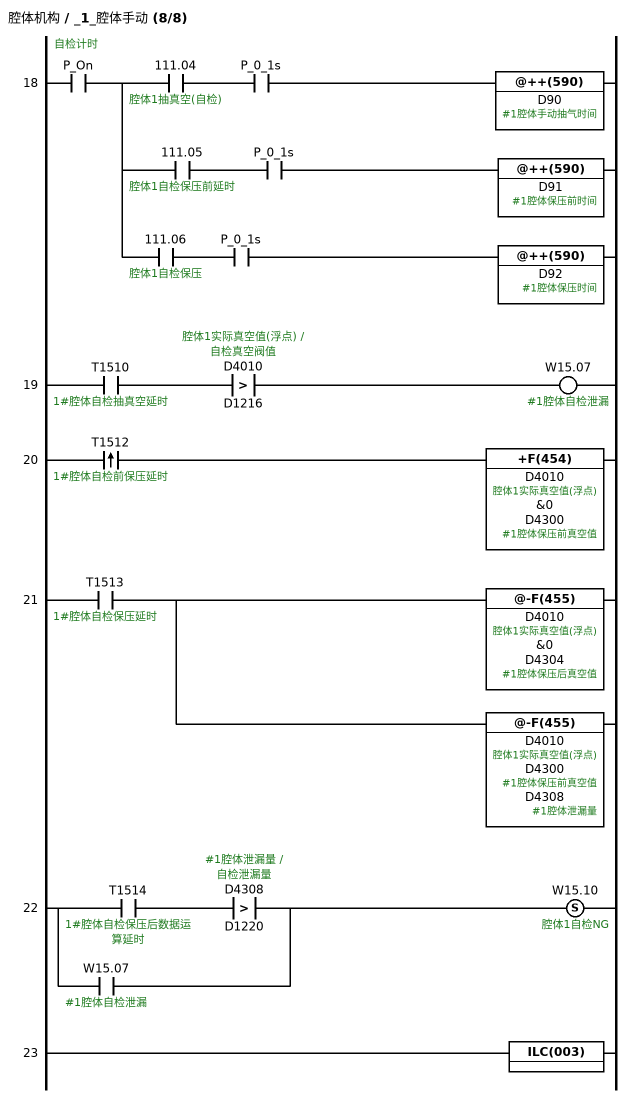
; rung 18: 自检计时
LD P_On
OUT TR0
AND 111.04  ; 腔体1抽真空(自检)
AND P_0_1s
@++(590) D90  ; #1腔体手动抽气时间
LD TR0
AND 111.05  ; 腔体1自检保压前延时
AND P_0_1s
@++(590) D91  ; #1腔体保压前时间
LD TR0
AND 111.06  ; 腔体1自检保压
AND P_0_1s
@++(590) D92  ; #1腔体保压时间
; rung 19
LD T1510  ; 1#腔体自检抽真空延时
AND>F(333) D4010 D1216  ; 腔体1实际真空值(浮点), 自检真空阀值
OUT W15.07  ; #1腔体自检泄漏
; rung 20
@LD T1512  ; 1#腔体自检前保压延时
+F(454) D4010 &0 D4300  ; 腔体1实际真空值(浮点), #1腔体保压前真空值
; rung 21
LD T1513  ; 1#腔体自检保压延时
@-F(455) D4010 &0 D4304  ; 腔体1实际真空值(浮点), #1腔体保压后真空值
@-F(455) D4010 D4300 D4308  ; 腔体1实际真空值(浮点), #1腔体保压前真空值, #1腔体泄漏量
; rung 22
LD T1514  ; 1#腔体自检保压后数据运算延时
AND>F(333) D4308 D1220  ; #1腔体泄漏量, 自检泄漏量
OR W15.07  ; #1腔体自检泄漏
SET W15.10  ; 腔体1自检NG
; rung 23
ILC(003)

### Section _2_腔体手动

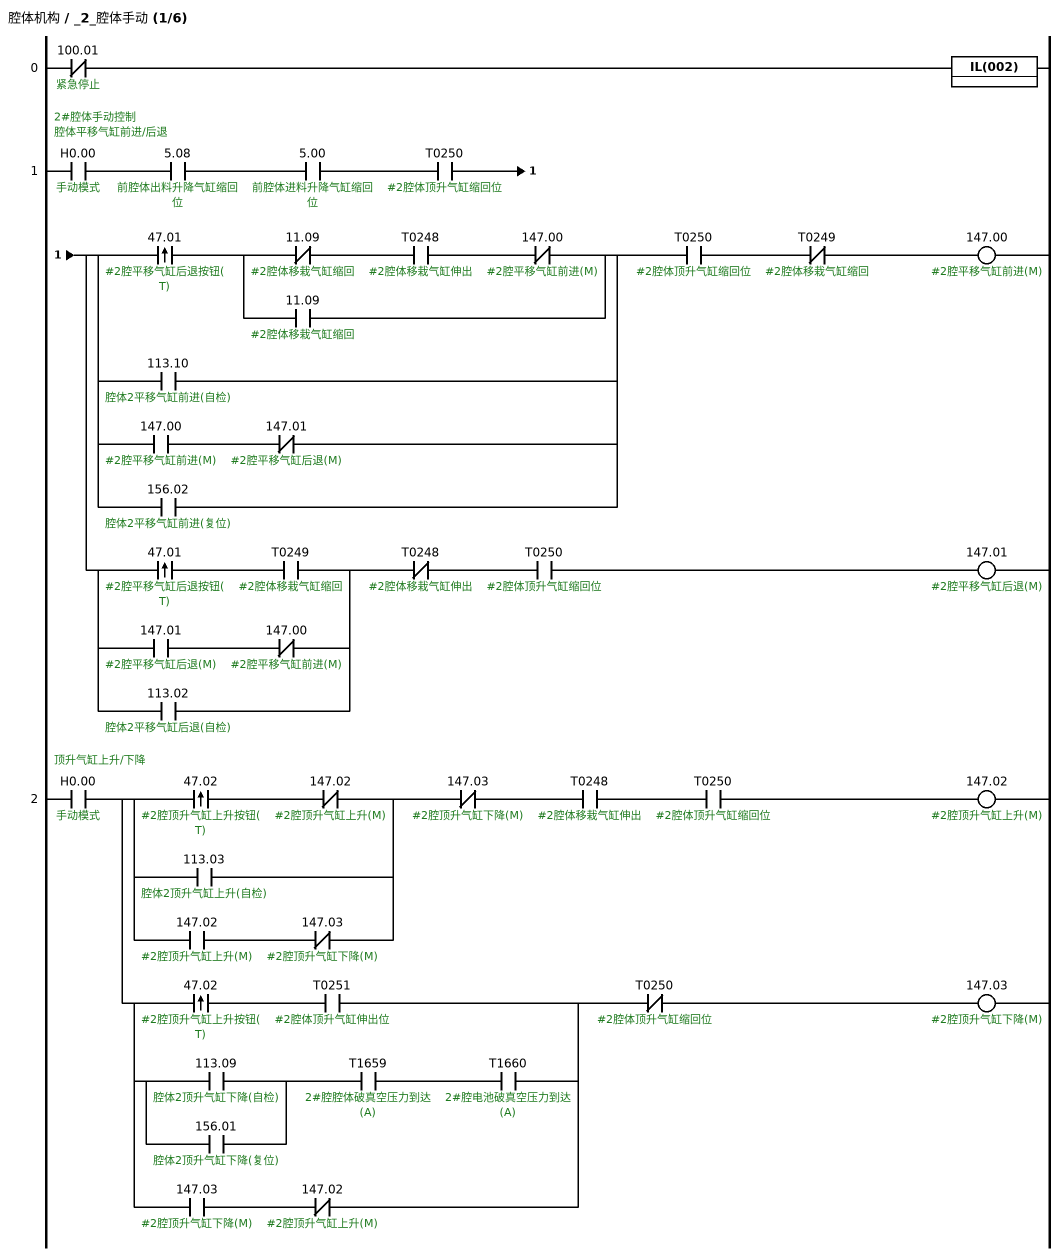
; rung 0
LDNOT 100.01  ; 紧急停止
IL(002)
; rung 1: 2#腔体手动控制 / 腔体平移气缸前进/后退
LD H0.00  ; 手动模式
AND 5.08  ; 前腔体出料升降气缸缩回位
AND 5.00  ; 前腔体进料升降气缸缩回位
AND T0250  ; #2腔体顶升气缸缩回位
OUT TR0
@LD 47.01  ; #2腔平移气缸后退按钮(T)
LDNOT 11.09  ; #2腔体移栽气缸缩回
AND T0248  ; #2腔体移栽气缸伸出
ANDNOT 147.00  ; #2腔平移气缸前进(M)
OR 11.09  ; #2腔体移栽气缸缩回
ANDLD
OR 113.10  ; 腔体2平移气缸前进(自检)
LD 147.00  ; #2腔平移气缸前进(M)
ANDNOT 147.01  ; #2腔平移气缸后退(M)
ORLD
OR 156.02  ; 腔体2平移气缸前进(复位)
ANDLD
AND T0250  ; #2腔体顶升气缸缩回位
ANDNOT T0249  ; #2腔体移栽气缸缩回
OUT 147.00  ; #2腔平移气缸前进(M)
LD TR0
@LD 47.01  ; #2腔平移气缸后退按钮(T)
AND T0249  ; #2腔体移栽气缸缩回
LD 147.01  ; #2腔平移气缸后退(M)
ANDNOT 147.00  ; #2腔平移气缸前进(M)
ORLD
OR 113.02  ; 腔体2平移气缸后退(自检)
ANDLD
ANDNOT T0248  ; #2腔体移栽气缸伸出
AND T0250  ; #2腔体顶升气缸缩回位
OUT 147.01  ; #2腔平移气缸后退(M)
; rung 2: 顶升气缸上升/下降
LD H0.00  ; 手动模式
OUT TR0
@LD 47.02  ; #2腔顶升气缸上升按钮(T)
ANDNOT 147.02  ; #2腔顶升气缸上升(M)
OR 113.03  ; 腔体2顶升气缸上升(自检)
LD 147.02  ; #2腔顶升气缸上升(M)
ANDNOT 147.03  ; #2腔顶升气缸下降(M)
ORLD
ANDLD
ANDNOT 147.03  ; #2腔顶升气缸下降(M)
AND T0248  ; #2腔体移栽气缸伸出
AND T0250  ; #2腔体顶升气缸缩回位
OUT 147.02  ; #2腔顶升气缸上升(M)
LD TR0
@LD 47.02  ; #2腔顶升气缸上升按钮(T)
AND T0251  ; #2腔体顶升气缸伸出位
LD 113.09  ; 腔体2顶升气缸下降(自检)
OR 156.01  ; 腔体2顶升气缸下降(复位)
AND T1659  ; 2#腔腔体破真空压力到达(A)
AND T1660  ; 2#腔电池破真空压力到达(A)
ORLD
LD 147.03  ; #2腔顶升气缸下降(M)
ANDNOT 147.02  ; #2腔顶升气缸上升(M)
ORLD
ANDLD
ANDNOT T0250  ; #2腔体顶升气缸缩回位
OUT 147.03  ; #2腔顶升气缸下降(M)

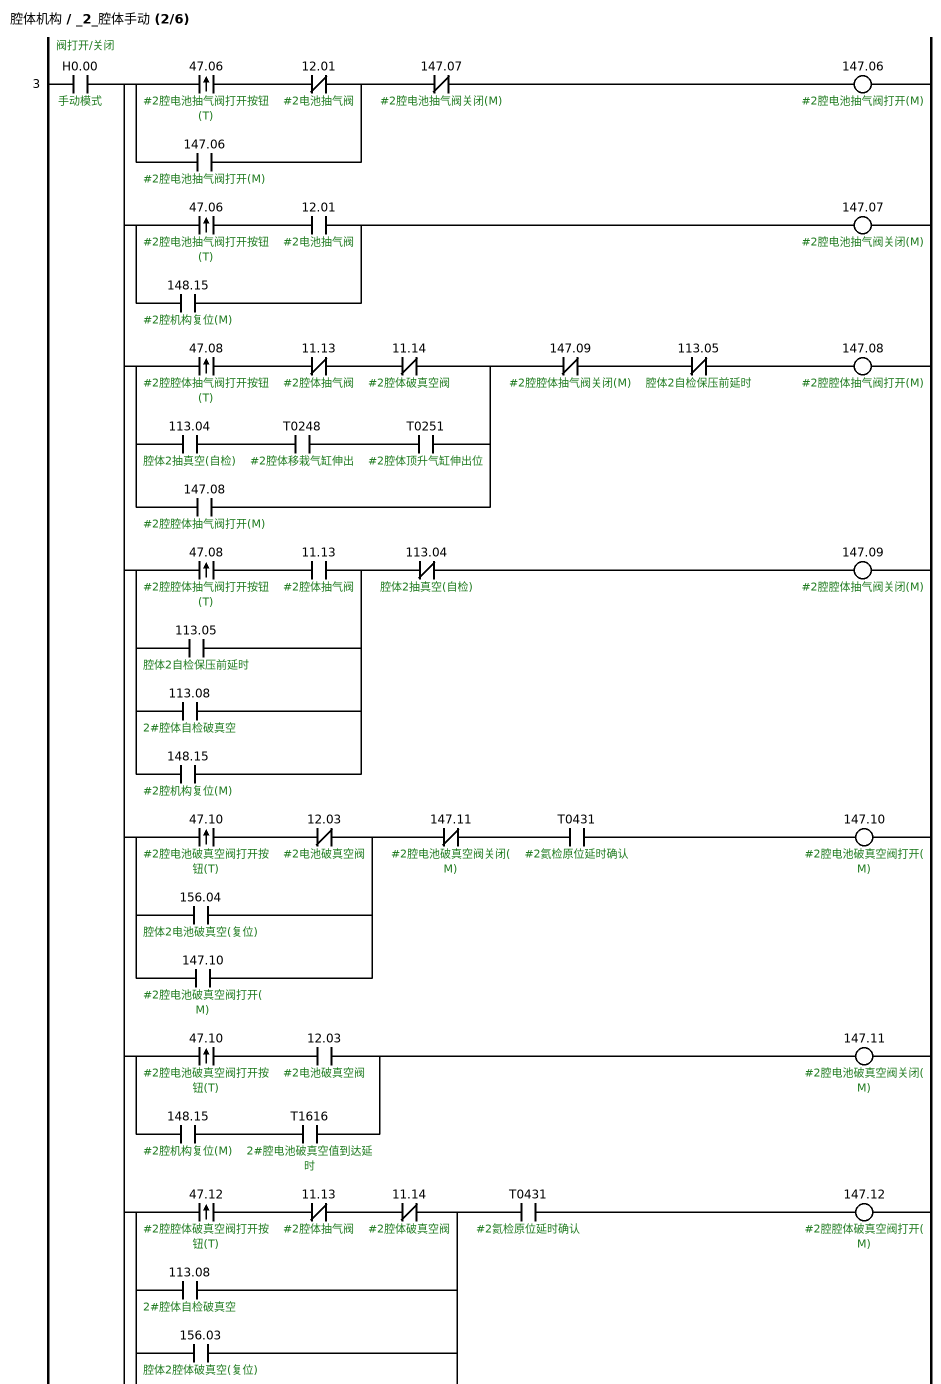

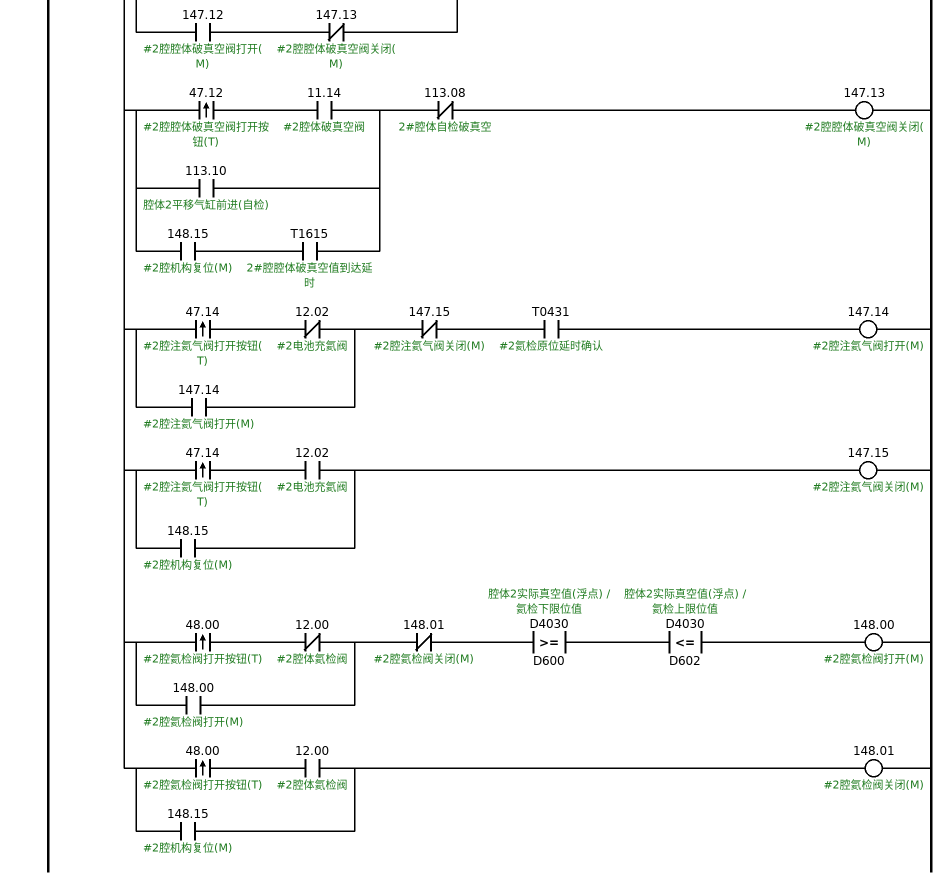
; rung 3: 阀打开/关闭
LD H0.00  ; 手动模式
OUT TR0
@LD 47.06  ; #2腔电池抽气阀打开按钮(T)
ANDNOT 12.01  ; #2电池抽气阀
OR 147.06  ; #2腔电池抽气阀打开(M)
ANDLD
ANDNOT 147.07  ; #2腔电池抽气阀关闭(M)
OUT 147.06  ; #2腔电池抽气阀打开(M)
LD TR0
@LD 47.06  ; #2腔电池抽气阀打开按钮(T)
AND 12.01  ; #2电池抽气阀
OR 148.15  ; #2腔机构复位(M)
ANDLD
OUT 147.07  ; #2腔电池抽气阀关闭(M)
LD TR0
@LD 47.08  ; #2腔腔体抽气阀打开按钮(T)
ANDNOT 11.13  ; #2腔体抽气阀
ANDNOT 11.14  ; #2腔体破真空阀
LD 113.04  ; 腔体2抽真空(自检)
AND T0248  ; #2腔体移栽气缸伸出
AND T0251  ; #2腔体顶升气缸伸出位
ORLD
OR 147.08  ; #2腔腔体抽气阀打开(M)
ANDLD
ANDNOT 147.09  ; #2腔腔体抽气阀关闭(M)
ANDNOT 113.05  ; 腔体2自检保压前延时
OUT 147.08  ; #2腔腔体抽气阀打开(M)
LD TR0
@LD 47.08  ; #2腔腔体抽气阀打开按钮(T)
AND 11.13  ; #2腔体抽气阀
OR 113.05  ; 腔体2自检保压前延时
OR 113.08  ; 2#腔体自检破真空
OR 148.15  ; #2腔机构复位(M)
ANDLD
ANDNOT 113.04  ; 腔体2抽真空(自检)
OUT 147.09  ; #2腔腔体抽气阀关闭(M)
LD TR0
@LD 47.10  ; #2腔电池破真空阀打开按钮(T)
ANDNOT 12.03  ; #2电池破真空阀
OR 156.04  ; 腔体2电池破真空(复位)
OR 147.10  ; #2腔电池破真空阀打开(M)
ANDLD
ANDNOT 147.11  ; #2腔电池破真空阀关闭(M)
AND T0431  ; #2氦检原位延时确认
OUT 147.10  ; #2腔电池破真空阀打开(M)
LD TR0
@LD 47.10  ; #2腔电池破真空阀打开按钮(T)
AND 12.03  ; #2电池破真空阀
LD 148.15  ; #2腔机构复位(M)
AND T1616  ; 2#腔电池破真空值到达延时
ORLD
ANDLD
OUT 147.11  ; #2腔电池破真空阀关闭(M)
LD TR0
@LD 47.12  ; #2腔腔体破真空阀打开按钮(T)
ANDNOT 11.13  ; #2腔体抽气阀
ANDNOT 11.14  ; #2腔体破真空阀
OR 113.08  ; 2#腔体自检破真空
OR 156.03  ; 腔体2腔体破真空(复位)
LD 147.12  ; #2腔腔体破真空阀打开(M)
ANDNOT 147.13  ; #2腔腔体破真空阀关闭(M)
ORLD
ANDLD
AND T0431  ; #2氦检原位延时确认
OUT 147.12  ; #2腔腔体破真空阀打开(M)
LD TR0
@LD 47.12  ; #2腔腔体破真空阀打开按钮(T)
AND 11.14  ; #2腔体破真空阀
OR 113.10  ; 腔体2平移气缸前进(自检)
LD 148.15  ; #2腔机构复位(M)
AND T1615  ; 2#腔腔体破真空值到达延时
ORLD
ANDLD
ANDNOT 113.08  ; 2#腔体自检破真空
OUT 147.13  ; #2腔腔体破真空阀关闭(M)
LD TR0
@LD 47.14  ; #2腔注氦气阀打开按钮(T)
ANDNOT 12.02  ; #2电池充氦阀
OR 147.14  ; #2腔注氦气阀打开(M)
ANDLD
ANDNOT 147.15  ; #2腔注氦气阀关闭(M)
AND T0431  ; #2氦检原位延时确认
OUT 147.14  ; #2腔注氦气阀打开(M)
LD TR0
@LD 47.14  ; #2腔注氦气阀打开按钮(T)
AND 12.02  ; #2电池充氦阀
OR 148.15  ; #2腔机构复位(M)
ANDLD
OUT 147.15  ; #2腔注氦气阀关闭(M)
LD TR0
@LD 48.00  ; #2腔氦检阀打开按钮(T)
ANDNOT 12.00  ; #2腔体氦检阀
OR 148.00  ; #2腔氦检阀打开(M)
ANDLD
ANDNOT 148.01  ; #2腔氦检阀关闭(M)
AND>=F(334) D4030 D600  ; 腔体2实际真空值(浮点), 氦检下限位值
AND<=F(332) D4030 D602  ; 腔体2实际真空值(浮点), 氦检上限位值
OUT 148.00  ; #2腔氦检阀打开(M)
LD TR0
@LD 48.00  ; #2腔氦检阀打开按钮(T)
AND 12.00  ; #2腔体氦检阀
OR 148.15  ; #2腔机构复位(M)
ANDLD
OUT 148.01  ; #2腔氦检阀关闭(M)

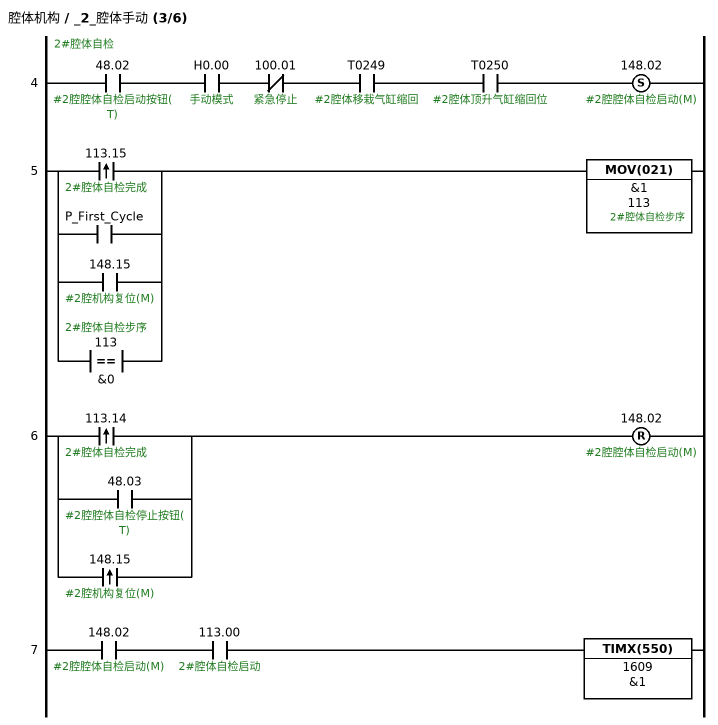
; rung 4: 2#腔体自检
LD 48.02  ; #2腔腔体自检启动按钮(T)
AND H0.00  ; 手动模式
ANDNOT 100.01  ; 紧急停止
AND T0249  ; #2腔体移栽气缸缩回
AND T0250  ; #2腔体顶升气缸缩回位
SET 148.02  ; #2腔腔体自检启动(M)
; rung 5
@LD 113.15  ; 2#腔体自检完成
OR P_First_Cycle
OR 148.15  ; #2腔机构复位(M)
OR=(300) 113 &0  ; 2#腔体自检步序
MOV(021) &1 113  ; 2#腔体自检步序
; rung 6
@LD 113.14  ; 2#腔体自检完成
OR 48.03  ; #2腔腔体自检停止按钮(T)
@OR 148.15  ; #2腔机构复位(M)
RSET 148.02  ; #2腔腔体自检启动(M)
; rung 7
LD 148.02  ; #2腔腔体自检启动(M)
AND 113.00  ; 2#腔体自检启动
TIMX(550) 1609 &1

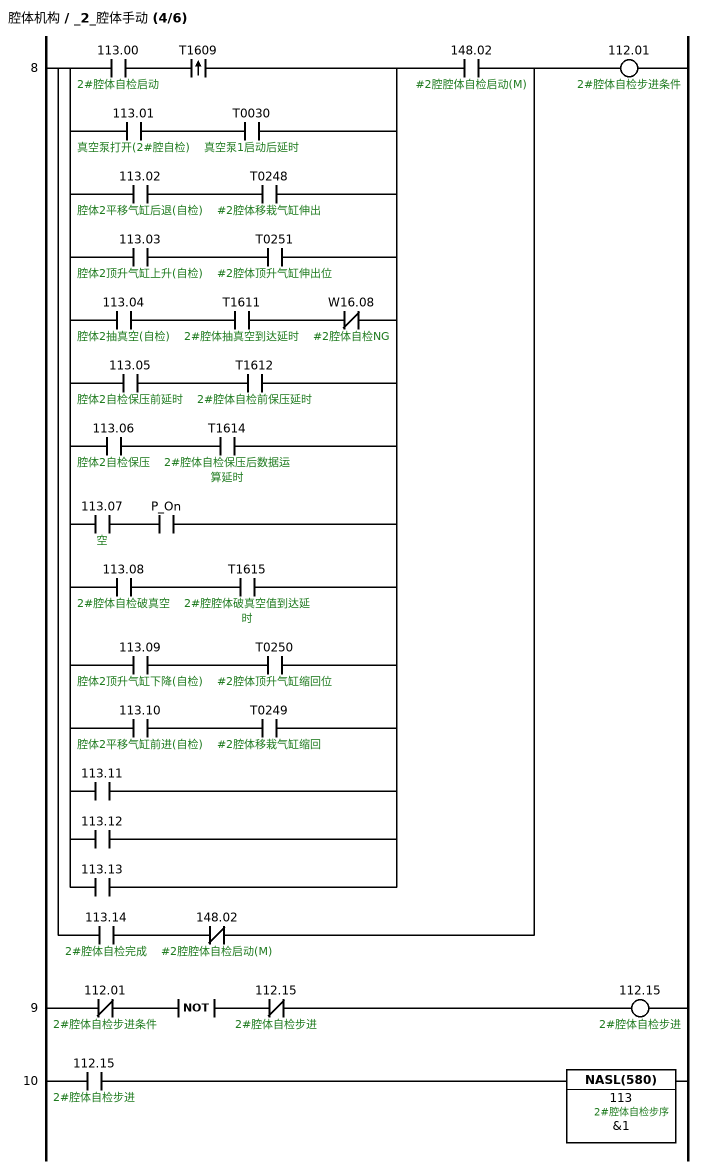
; rung 8
LD 113.00  ; 2#腔体自检启动
@AND T1609
LD 113.01  ; 真空泵打开(2#腔自检)
AND T0030  ; 真空泵1启动后延时
ORLD
LD 113.02  ; 腔体2平移气缸后退(自检)
AND T0248  ; #2腔体移栽气缸伸出
ORLD
LD 113.03  ; 腔体2顶升气缸上升(自检)
AND T0251  ; #2腔体顶升气缸伸出位
ORLD
LD 113.04  ; 腔体2抽真空(自检)
AND T1611  ; 2#腔体抽真空到达延时
ANDNOT W16.08  ; #2腔体自检NG
ORLD
LD 113.05  ; 腔体2自检保压前延时
AND T1612  ; 2#腔体自检前保压延时
ORLD
LD 113.06  ; 腔体2自检保压
AND T1614  ; 2#腔体自检保压后数据运算延时
ORLD
LD 113.07  ; 空
AND P_On
ORLD
LD 113.08  ; 2#腔体自检破真空
AND T1615  ; 2#腔腔体破真空值到达延时
ORLD
LD 113.09  ; 腔体2顶升气缸下降(自检)
AND T0250  ; #2腔体顶升气缸缩回位
ORLD
LD 113.10  ; 腔体2平移气缸前进(自检)
AND T0249  ; #2腔体移栽气缸缩回
ORLD
OR 113.11
OR 113.12
OR 113.13
AND 148.02  ; #2腔腔体自检启动(M)
LD 113.14  ; 2#腔体自检完成
ANDNOT 148.02  ; #2腔腔体自检启动(M)
ORLD
OUT 112.01  ; 2#腔体自检步进条件
; rung 9
LDNOT 112.01  ; 2#腔体自检步进条件
NOT(520)
ANDNOT 112.15  ; 2#腔体自检步进
OUT 112.15  ; 2#腔体自检步进
; rung 10
LD 112.15  ; 2#腔体自检步进
NASL(580) 113 &1  ; 2#腔体自检步序

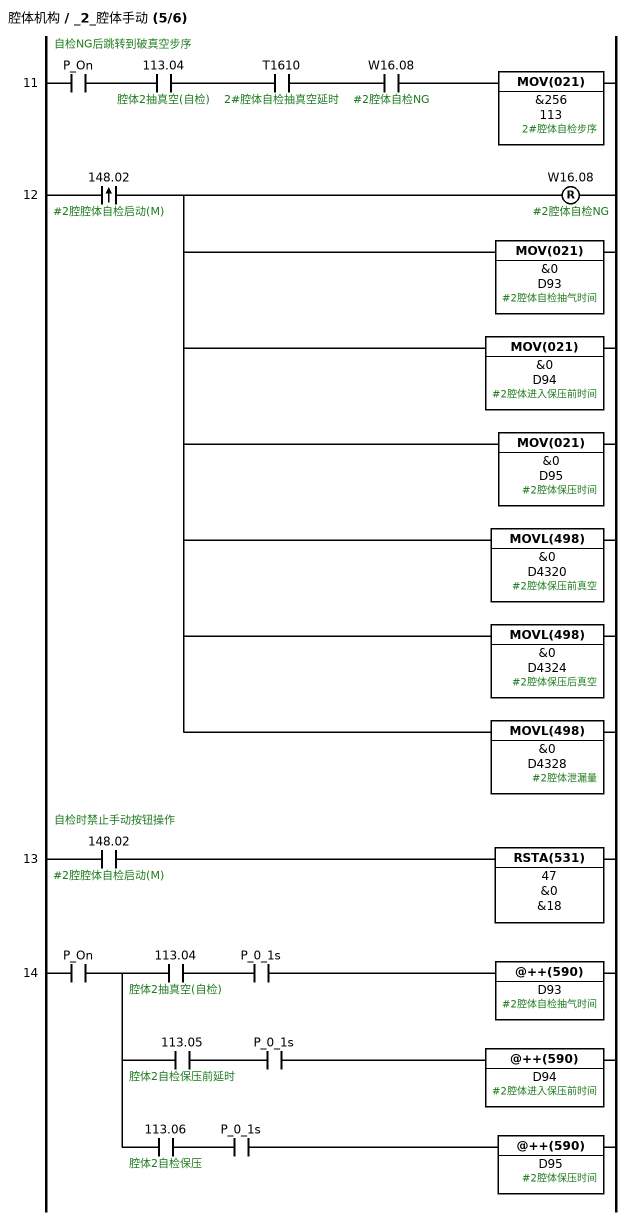
; rung 11: 自检NG后跳转到破真空步序
LD P_On
AND 113.04  ; 腔体2抽真空(自检)
AND T1610  ; 2#腔体自检抽真空延时
AND W16.08  ; #2腔体自检NG
MOV(021) &256 113  ; 2#腔体自检步序
; rung 12
@LD 148.02  ; #2腔腔体自检启动(M)
RSET W16.08  ; #2腔体自检NG
MOV(021) &0 D93  ; #2腔体自检抽气时间
MOV(021) &0 D94  ; #2腔体进入保压前时间
MOV(021) &0 D95  ; #2腔体保压时间
MOVL(498) &0 D4320  ; #2腔体保压前真空
MOVL(498) &0 D4324  ; #2腔体保压后真空
MOVL(498) &0 D4328  ; #2腔体泄漏量
; rung 13: 自检时禁止手动按钮操作
LD 148.02  ; #2腔腔体自检启动(M)
RSTA(531) 47 &0 &18
; rung 14
LD P_On
OUT TR0
AND 113.04  ; 腔体2抽真空(自检)
AND P_0_1s
@++(590) D93  ; #2腔体自检抽气时间
LD TR0
AND 113.05  ; 腔体2自检保压前延时
AND P_0_1s
@++(590) D94  ; #2腔体进入保压前时间
LD TR0
AND 113.06  ; 腔体2自检保压
AND P_0_1s
@++(590) D95  ; #2腔体保压时间

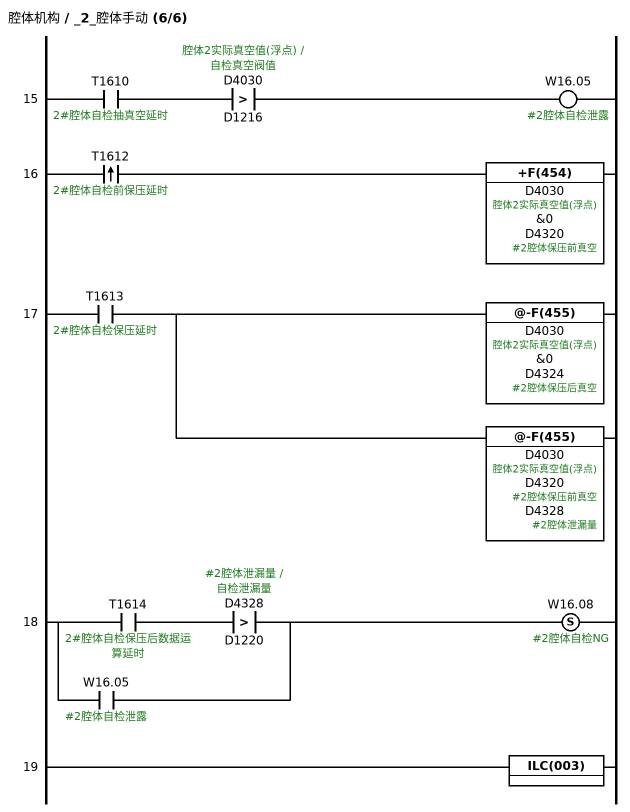
; rung 15
LD T1610  ; 2#腔体自检抽真空延时
AND>F(333) D4030 D1216  ; 腔体2实际真空值(浮点), 自检真空阀值
OUT W16.05  ; #2腔体自检泄露
; rung 16
@LD T1612  ; 2#腔体自检前保压延时
+F(454) D4030 &0 D4320  ; 腔体2实际真空值(浮点), #2腔体保压前真空
; rung 17
LD T1613  ; 2#腔体自检保压延时
@-F(455) D4030 &0 D4324  ; 腔体2实际真空值(浮点), #2腔体保压后真空
@-F(455) D4030 D4320 D4328  ; 腔体2实际真空值(浮点), #2腔体保压前真空, #2腔体泄漏量
; rung 18
LD T1614  ; 2#腔体自检保压后数据运算延时
AND>F(333) D4328 D1220  ; #2腔体泄漏量, 自检泄漏量
OR W16.05  ; #2腔体自检泄露
SET W16.08  ; #2腔体自检NG
; rung 19
ILC(003)

### Section _3_腔体手动

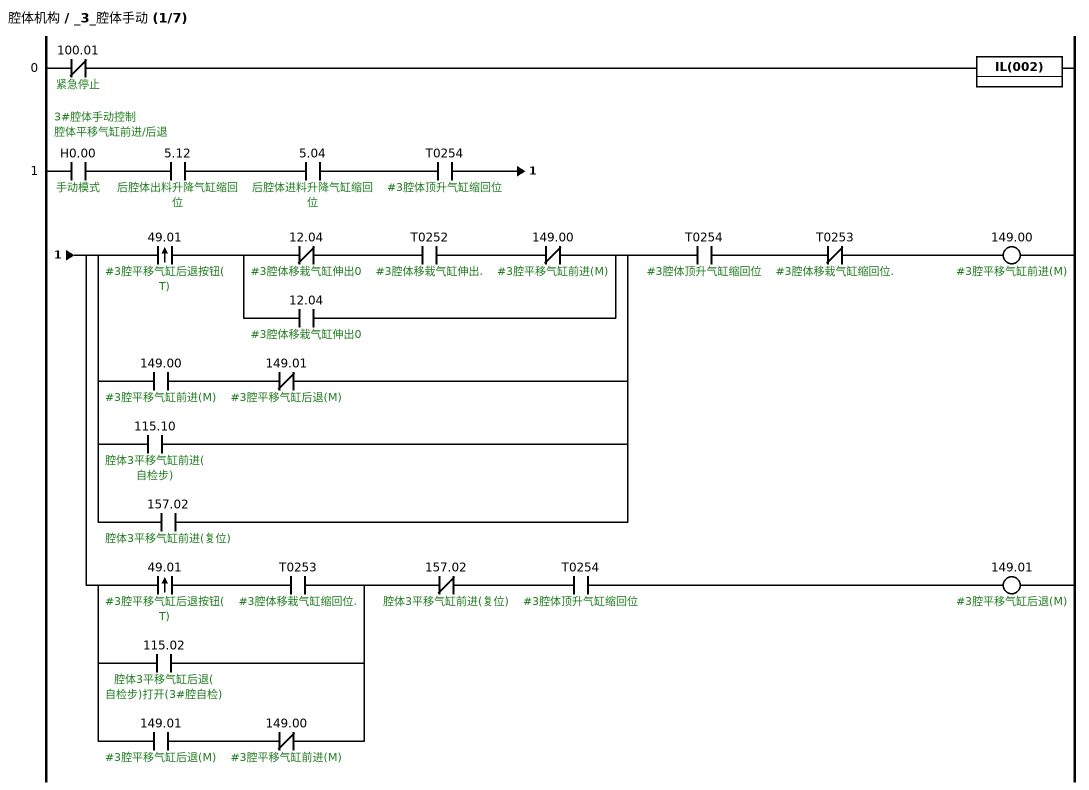
; rung 0
LDNOT 100.01  ; 紧急停止
IL(002)
; rung 1: 3#腔体手动控制 / 腔体平移气缸前进/后退
LD H0.00  ; 手动模式
AND 5.12  ; 后腔体出料升降气缸缩回位
AND 5.04  ; 后腔体进料升降气缸缩回位
AND T0254  ; #3腔体顶升气缸缩回位
OUT TR0
@LD 49.01  ; #3腔平移气缸后退按钮(T)
LDNOT 12.04  ; #3腔体移栽气缸伸出0
AND T0252  ; #3腔体移栽气缸伸出.
ANDNOT 149.00  ; #3腔平移气缸前进(M)
OR 12.04  ; #3腔体移栽气缸伸出0
ANDLD
LD 149.00  ; #3腔平移气缸前进(M)
ANDNOT 149.01  ; #3腔平移气缸后退(M)
ORLD
OR 115.10  ; 腔体3平移气缸前进(自检步)
OR 157.02  ; 腔体3平移气缸前进(复位)
ANDLD
AND T0254  ; #3腔体顶升气缸缩回位
ANDNOT T0253  ; #3腔体移栽气缸缩回位.
OUT 149.00  ; #3腔平移气缸前进(M)
LD TR0
@LD 49.01  ; #3腔平移气缸后退按钮(T)
AND T0253  ; #3腔体移栽气缸缩回位.
OR 115.02  ; 腔体3平移气缸后退(自检步)打开(3#腔自检)
LD 149.01  ; #3腔平移气缸后退(M)
ANDNOT 149.00  ; #3腔平移气缸前进(M)
ORLD
ANDLD
ANDNOT 157.02  ; 腔体3平移气缸前进(复位)
AND T0254  ; #3腔体顶升气缸缩回位
OUT 149.01  ; #3腔平移气缸后退(M)

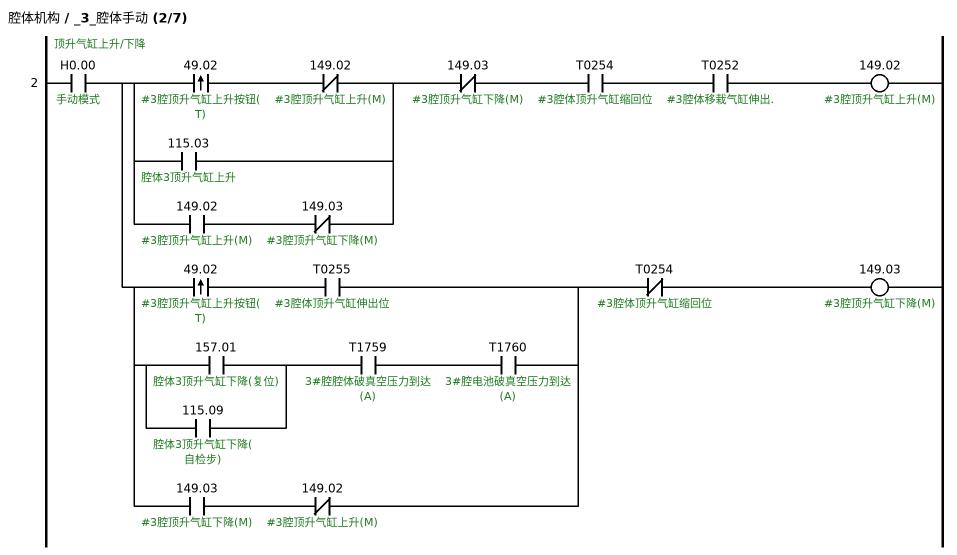
; rung 2: 顶升气缸上升/下降
LD H0.00  ; 手动模式
OUT TR0
@LD 49.02  ; #3腔顶升气缸上升按钮(T)
ANDNOT 149.02  ; #3腔顶升气缸上升(M)
OR 115.03  ; 腔体3顶升气缸上升
LD 149.02  ; #3腔顶升气缸上升(M)
ANDNOT 149.03  ; #3腔顶升气缸下降(M)
ORLD
ANDLD
ANDNOT 149.03  ; #3腔顶升气缸下降(M)
AND T0254  ; #3腔体顶升气缸缩回位
AND T0252  ; #3腔体移栽气缸伸出.
OUT 149.02  ; #3腔顶升气缸上升(M)
LD TR0
@LD 49.02  ; #3腔顶升气缸上升按钮(T)
AND T0255  ; #3腔体顶升气缸伸出位
LD 157.01  ; 腔体3顶升气缸下降(复位)
OR 115.09  ; 腔体3顶升气缸下降(自检步)
AND T1759  ; 3#腔腔体破真空压力到达(A)
AND T1760  ; 3#腔电池破真空压力到达(A)
ORLD
LD 149.03  ; #3腔顶升气缸下降(M)
ANDNOT 149.02  ; #3腔顶升气缸上升(M)
ORLD
ANDLD
ANDNOT T0254  ; #3腔体顶升气缸缩回位
OUT 149.03  ; #3腔顶升气缸下降(M)

